// TIA Portal project "level-controle-factoryIO" (V17)

(* hardware
DEVICE "S71500/ET200MP-Station_1"  S7-1500 station
   slot 0: "Profilschiene_0"  6ES7 590-1***0-0AA0
   slot 1: "PLC_1"  CPU 1511-1 PN  6ES7 511-1AK00-0AB0  V1.8
   slot 2: "AI 8xU/I/RTD/TC ST_1"  AI 8xU/I/RTD/TC ST  6ES7 531-7KF00-0AB0  V2.0
   slot 3: "AI 8xU/I/RTD/TC ST_2"  AI 8xU/I/RTD/TC ST  6ES7 531-7KF00-0AB0  V2.0
   slot 4: "AI 8xU/I/RTD/TC ST_3"  AI 8xU/I/RTD/TC ST  6ES7 531-7KF00-0AB0  V2.0
   slot 5: "AI 8xU/I/RTD/TC ST_4"  AI 8xU/I/RTD/TC ST  6ES7 531-7KF00-0AB0  V2.0
   slot 6: "DI 16x24VDC BA_1"  DI 16x24VDC BA  6ES7 521-1BH10-0AA0  V1.0
DEVICE "HMI_1"  KTP900 Basic PN
   slot 0: "HMI_1"  KTP900 Basic PN  6AV2 123-2JB03-0AX0  17.0.0.0
   slot 1: "HMI_RT_1"  KTP900 Basic PN  6AV2 123-2JB03-0AX0  17.0.0.0
   slot 5: "HMI_1.IE_CP_1"  PROFINET Interface  17.0.0.0
      slot 1: "PROFINET Interface_1"  PROFINET Interface
         slot 1: "Port_1"  Port
*)

// ===== PLC "PLC_1"  CPU 1511-1 PN =====

VAR_GLOBAL   // PLC tag table "Standard-Variablentabelle"
   "Clock_Byte" AT %MB0 : Byte;
   "Clock_10Hz" AT %M0.0 : Bool;
   "Clock_5Hz" AT %M0.1 : Bool;
   "Clock_2.5Hz" AT %M0.2 : Bool;
   "Clock_2Hz" AT %M0.3 : Bool;
   "Clock_1.25Hz" AT %M0.4 : Bool;
   "Clock_1Hz" AT %M0.5 : Bool;
   "Clock_0.625Hz" AT %M0.6 : Bool;
   "Clock_0.5Hz" AT %M0.7 : Bool;
   "System_Byte" AT %MB1 : Byte;
   "FirstScan" AT %M1.0 : Bool;
   "DiagStatusUpdate" AT %M1.1 : Bool;
   "AlwaysTRUE" AT %M1.2 : Bool;
   "AlwaysFALSE" AT %M1.3 : Bool;
   "Tag_1" AT %M110.0 : Bool;
END_VAR

VAR_GLOBAL   // PLC tag table "Input"
   "I_LevelMeter" AT %ID30 : Real;
   "I_FlowMeter" AT %ID34 : Real;
   "I_FactoryRuning" AT %I0.0 : Bool;
END_VAR

VAR_GLOBAL   // PLC tag table "Output"
   "O_FillValve" AT %QD30 : Real;
   "O_DischargeValve" AT %QD34 : Real;
   "O_Empty" AT %Q0.0 : Bool;
END_VAR

// folder: 00_Visu

DATA_BLOCK "VisuData"   // DB9
{ S7_Optimized_Access := 'TRUE' }
VERSION : 0.1
   VAR
      Start : Bool;
      Stop : Bool;
      Empty : Bool;
      Controller : Int;
      RandomDisturbance : Int;
      SetPoint : Real;
      Outflow : Real;
      LevelMeterShow : Real;
      SetPointShow : Real;
      FillValveShow : Real;
      TopPump : Int;
      LowPump : Int;
      Status : Bool;
      default : Bool;
      finish_training : Int;
      factoryio_connect : Bool;
   END_VAR
BEGIN
END_DATA_BLOCK

// folder: 01_Convert

DATA_BLOCK "ConvertData"   // DB4
{ S7_Optimized_Access := 'TRUE' }
VERSION : 0.1
   VAR
      SetPoint10 : Real;
   END_VAR
BEGIN
END_DATA_BLOCK

// folder: 02_Controller

DATA_BLOCK "ControllerData"   // DB1
{ S7_Optimized_Access := 'TRUE' }
VERSION : 0.1
   VAR
      PID_Compact : Bool;
      Output_PID_Compact : Real;
      "IMC+PID" : Bool;
      rate : Real;
      hysteresis : Real;
      kp : Real;
      ki : Real;
      kd : Real;
   END_VAR
BEGIN
END_DATA_BLOCK

// folder: 02_Controller/NeuralNetwork

DATA_BLOCK "NeuroData"   // DB18
{ S7_Optimized_Access := 'TRUE' }
VERSION : 0.1
   VAR
      finish_measurment : Bool;
      disturbance : Real;
      PV : Real;
      MV : Real;
      SP : Real;
      stop_training_inw : Bool;
      stop_training_mod : Bool;
      epoka : Real;
      error_ep_m : Real;
      error_ep_i : Real;
      error_stop_m : Real;
      error_stop_i : Real;
      epoka_m : Real;
      epoka_i : Real;
      move : Bool;
      p_move : Bool;
      finish_training : Bool;
   END_VAR
BEGIN
END_DATA_BLOCK

// folder: System blocks/Program resources

DATA_BLOCK "PID_DB"   // DB2
{ S7_Optimized_Access := 'FALSE' }
VERSION : 0.1
// stored: InstanceOfName PID
"PID"
BEGIN
END_DATA_BLOCK

DATA_BLOCK "RandomDisturbance_DB"   // DB5
{ S7_Optimized_Access := 'TRUE' }
VERSION : 0.1
// stored: InstanceOfName RandomDisturbance
"RandomDisturbance"
BEGIN
END_DATA_BLOCK

DATA_BLOCK "RAMP_DB"   // DB6
{ S7_Optimized_Access := 'TRUE' }
VERSION : 0.1
// stored: InstanceOfName RAMP
"RAMP"
BEGIN
END_DATA_BLOCK

DATA_BLOCK "RegSugeno_DB"   // DB7
{ S7_Optimized_Access := 'TRUE' }
VERSION : 0.1
// stored: InstanceOfName Takagi-SugenoFuzzy-PI
"Takagi-SugenoFuzzy-PI"
BEGIN
END_DATA_BLOCK

DATA_BLOCK "Training_DB"   // DB10
{ S7_Optimized_Access := 'FALSE' }
VERSION : 0.1
// stored: InstanceOfName Training
"Training"
BEGIN
END_DATA_BLOCK

DATA_BLOCK "PID_DB_1"   // DB11
{ S7_Optimized_Access := 'FALSE' }
VERSION : 0.1
// stored: InstanceOfName PID
"PID"
BEGIN
END_DATA_BLOCK

DATA_BLOCK "Measurement_DB"   // DB12
{ S7_Optimized_Access := 'FALSE' }
VERSION : 0.1
// stored: InstanceOfName Measurement
"Measurement"
BEGIN
END_DATA_BLOCK

DATA_BLOCK "Object_DB"   // DB13
{ S7_Optimized_Access := 'FALSE' }
VERSION : 0.1
// stored: InstanceOfName Object
"Object"
BEGIN
END_DATA_BLOCK

DATA_BLOCK "Generator_DB"   // DB14
{ S7_Optimized_Access := 'FALSE' }
VERSION : 0.1
// stored: InstanceOfName Generator
"Generator"
BEGIN
END_DATA_BLOCK

DATA_BLOCK "IMC+PID_DB"   // DB15
{ S7_Optimized_Access := 'FALSE' }
VERSION : 0.1
// stored: InstanceOfName IMC+PID
"IMC+PID"
BEGIN
END_DATA_BLOCK

DATA_BLOCK "Model_DB"   // DB16
{ S7_Optimized_Access := 'FALSE' }
VERSION : 0.1
// stored: InstanceOfName Model
"Model"
BEGIN
END_DATA_BLOCK

DATA_BLOCK "Inversion_DB"   // DB17
{ S7_Optimized_Access := 'FALSE' }
VERSION : 0.1
// stored: InstanceOfName Inversion
"Inversion"
BEGIN
END_DATA_BLOCK

DATA_BLOCK "StartStop_DB"   // DB19
{ S7_Optimized_Access := 'TRUE' }
VERSION : 0.1
// stored: InstanceOfName StartStop
"StartStop"
BEGIN
END_DATA_BLOCK

DATA_BLOCK "On-Off_DB"   // DB20
{ S7_Optimized_Access := 'TRUE' }
VERSION : 0.1
// stored: InstanceOfName On-Off
"On-Off"
BEGIN
END_DATA_BLOCK

// folder: (top level)

FUNCTION "MHJ-PLC-Lab-Function-S71500" : Void   // FC9000, SCL
{ S7_Optimized_Access := 'TRUE' }
VERSION : 0.1
   VAR_TEMP
      Value : Byte;
      ForCounter : Int;
   END_VAR
   VAR CONSTANT
      Value_01_DW : DWord := 16#1223_5486;
      Value_02_DW : DWord := 16#A6C9_D1F5;
   END_VAR
BEGIN

   #Value:=PEEK(area := 16#82,
        dbNumber := 0,
        byteOffset := 511);
   #Value := #Value + 1;

   POKE(area := 16#82,
        dbNumber := 0,
        byteOffset := 511,
        value := #Value);

   POKE(area := 16#82,
        dbNumber := 0,
        byteOffset := 1016,
        value := #Value_01_DW);
   POKE(area := 16#82,
        dbNumber := 0,
        byteOffset := 1020,
        value := #Value_02_DW);

   FOR #ForCounter := 0 TO 63 DO
       #Value:=PEEK(area := 16#1,
            dbNumber := 0,
            byteOffset := #ForCounter);
       POKE(area := 16#81,
            dbNumber := 0,
            byteOffset := #ForCounter,
            value := #Value);
   END_FOR;
   #Value := PEEK(area := 16#1,
                  dbNumber := 0,
                  byteOffset := 512);
   POKE(area := 16#82,
        dbNumber := 0,
        byteOffset := 512,
        value := #Value);
END_FUNCTION

ORGANIZATION_BLOCK "Main"   // OB1, LAD, ProgramCycle
TITLE = "Main Program Sweep (Cycle)"
{ S7_Optimized_Access := 'TRUE' }
VERSION : 0.1
   VAR_INPUT
      Initial_Call : Bool;   // Initial call of this OB
      Remanence : Bool;   // =True, if remanent data are available
   END_VAR
BEGIN

REGION Network 1: Call: MHJ-PLC-Lab-Function-S71500
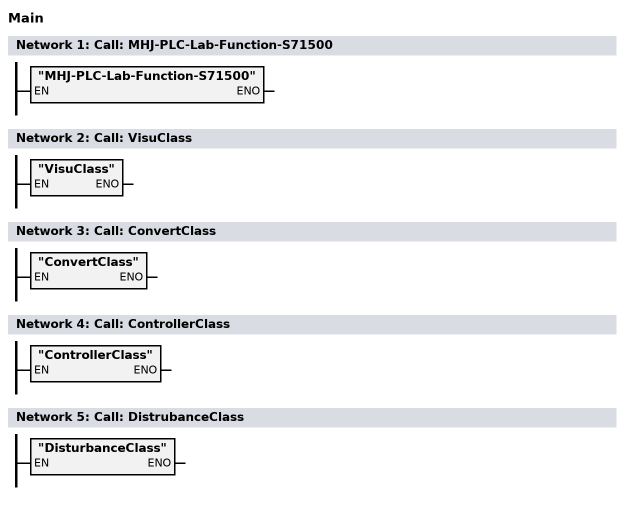
   RUNG wire#powerrail
      "MHJ-PLC-Lab-Function-S71500"()
   END_RUNG
   // the same network as SCL:
   "MHJ-PLC-Lab-Function-S71500"();
END_REGION

REGION Network 2: Call: VisuClass
   RUNG wire#powerrail
      "VisuClass"()
   END_RUNG
   // the same network as SCL:
   "VisuClass"();
END_REGION

REGION Network 3: Call: ConvertClass
   RUNG wire#powerrail
      "ConvertClass"()
   END_RUNG
   // the same network as SCL:
   "ConvertClass"();
END_REGION

REGION Network 4: Call: ControllerClass
   RUNG wire#powerrail
      "ControllerClass"()
   END_RUNG
   // the same network as SCL:
   "ControllerClass"();
END_REGION

REGION Network 5: Call: DistrubanceClass
   RUNG wire#powerrail
      "DisturbanceClass"()
   END_RUNG
   // the same network as SCL:
   "DisturbanceClass"();
END_REGION
END_ORGANIZATION_BLOCK

ORGANIZATION_BLOCK "Startup"   // OB100, LAD, Startup
TITLE = "Complete Restart"
{ S7_Optimized_Access := 'TRUE' }
VERSION : 0.1
   VAR_INPUT
      LostRetentive : Bool;   // True if retentive data are lost
      LostRTC : Bool;   // True if date and time are lost
   END_VAR
BEGIN

REGION Network 1: Call: StartupValues
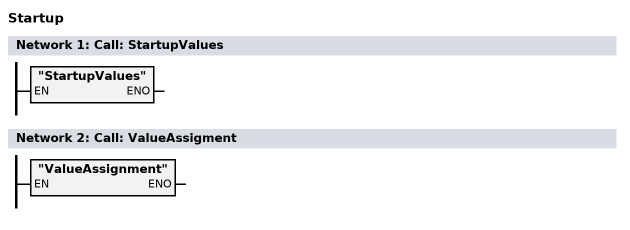
   RUNG wire#powerrail
      "StartupValues"()
   END_RUNG
   // the same network as SCL:
   "StartupValues"();
END_REGION

REGION Network 2: Call: ValueAssigment
   RUNG wire#powerrail
      "ValueAssignment"()
   END_RUNG
   // the same network as SCL:
   "ValueAssignment"();
END_REGION
END_ORGANIZATION_BLOCK

// folder: 00_Visu

FUNCTION "ShowPompOn" : Void   // FC6, LAD
TITLE = ShowPompOn
{ S7_Optimized_Access := 'TRUE' }
VERSION : 0.1
   VAR_TEMP   // added for the SCL form of the ladder/FBD networks
      _w1 : Bool;
   END_VAR
BEGIN

REGION Network 1: Move: TopPump
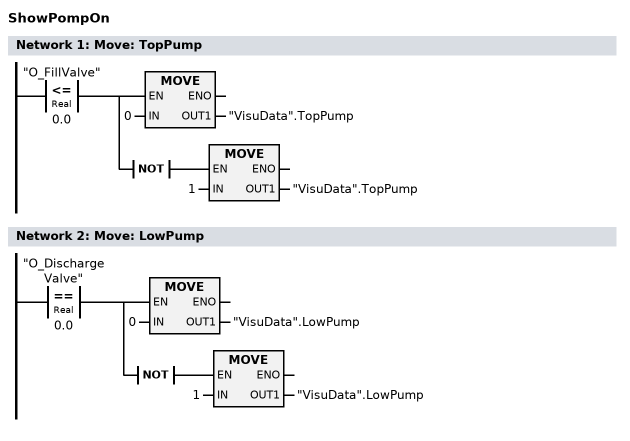
   RUNG wire#powerrail
      { S7_Templates := "SrcType := Real" } LE_Contact(in1 := "O_FillValve", in2 := 0.0)
      wire#w1
      Move(in := 0, out1 => "VisuData".TopPump)
   END_RUNG
   RUNG wire#w1
      Not()
      Move(in := 1, out1 => "VisuData".TopPump)
   END_RUNG
   // the same network as SCL:
   #_w1 := "O_FillValve" <= 0.0;
   IF #_w1 THEN "VisuData".TopPump := 0; END_IF;
   IF NOT #_w1 THEN "VisuData".TopPump := 1; END_IF;
END_REGION

REGION Network 2: Move: LowPump
   RUNG wire#powerrail
      { S7_Templates := "SrcType := Real" } EQ_Contact(in1 := "O_DischargeValve", in2 := 0.0)
      wire#w1
      Move(in := 0, out1 => "VisuData".LowPump)
   END_RUNG
   RUNG wire#w1
      Not()
      Move(in := 1, out1 => "VisuData".LowPump)
   END_RUNG
   // the same network as SCL:
   #_w1 := "O_DischargeValve" = 0.0;
   IF #_w1 THEN "VisuData".LowPump := 0; END_IF;
   IF NOT #_w1 THEN "VisuData".LowPump := 1; END_IF;
END_REGION
END_FUNCTION

FUNCTION "VisuClass" : Void   // FC8, LAD
TITLE = VisuClass
{ S7_Optimized_Access := 'TRUE' }
VERSION : 0.1
BEGIN

REGION Network 1: Call: StartStop
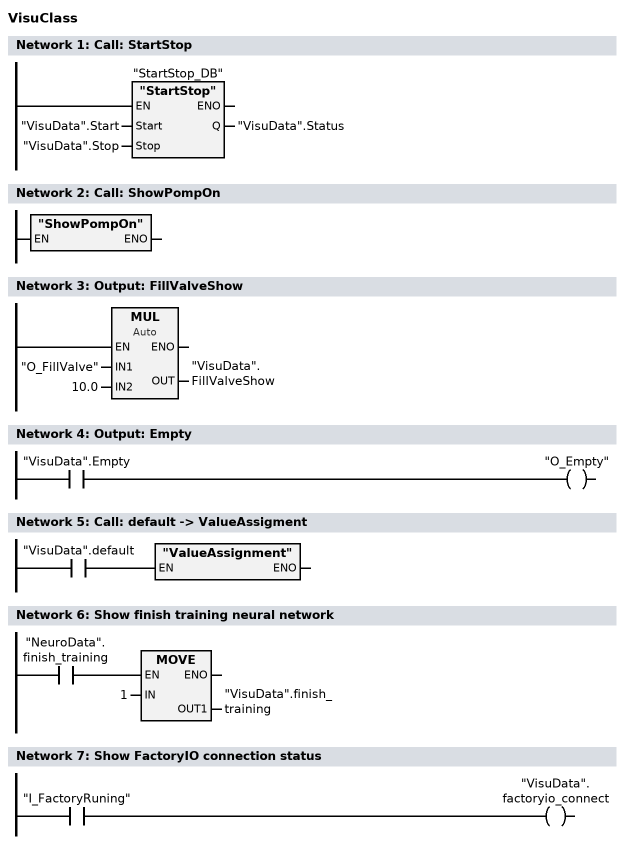
   RUNG wire#powerrail
      "StartStop_DB"(Start := "VisuData".Start, Stop := "VisuData".Stop, Q => "VisuData".Status)
   END_RUNG
   // the same network as SCL:
   "StartStop_DB"(Start := "VisuData".Start, Stop := "VisuData".Stop, Q => "VisuData".Status);   // "StartStop"
END_REGION

REGION Network 2: Call: ShowPompOn
   RUNG wire#powerrail
      "ShowPompOn"()
   END_RUNG
   // the same network as SCL:
   "ShowPompOn"();
END_REGION

REGION Network 3: Output: FillValveShow
   RUNG wire#powerrail
      Mul(in1 := "O_FillValve", in2 := 10.0, out => "VisuData".FillValveShow)
   END_RUNG
   // the same network as SCL:
   "VisuData".FillValveShow := "O_FillValve" * 10.0;
END_REGION

REGION Network 4: Output: Empty
   RUNG wire#powerrail
      Contact( "VisuData".Empty )
      Coil( "O_Empty" )
   END_RUNG
   // the same network as SCL:
   "O_Empty" := "VisuData".Empty;
END_REGION

REGION Network 5: Call: default -> ValueAssigment
   RUNG wire#powerrail
      Contact( "VisuData".default )
      "ValueAssignment"()
   END_RUNG
   // the same network as SCL:
   IF "VisuData".default THEN "ValueAssignment"(); END_IF;
END_REGION

REGION Network 6: Show finish training neural network
   RUNG wire#powerrail
      Contact( "NeuroData".finish_training )
      Move(in := 1, out1 => "VisuData".finish_training)
   END_RUNG
   // the same network as SCL:
   IF "NeuroData".finish_training THEN "VisuData".finish_training := 1; END_IF;
END_REGION

REGION Network 7: Show FactoryIO connection status
   RUNG wire#powerrail
      Contact( "I_FactoryRuning" )
      Coil( "VisuData".factoryio_connect )
   END_RUNG
   // the same network as SCL:
   "VisuData".factoryio_connect := "I_FactoryRuning";
END_REGION
END_FUNCTION

// folder: 01_Convert

FUNCTION "ConvertClass" : Void   // FC3, LAD
TITLE = ConvertClass
{ S7_Optimized_Access := 'TRUE' }
VERSION : 0.1
   VAR_TEMP
      Output_PID_Real : Real;
      PV : Real;
      SP : Real;
      SPRamp : Real;
   END_VAR
BEGIN

REGION Network 1: Convert SetPoint: 0-300 -> 0-10
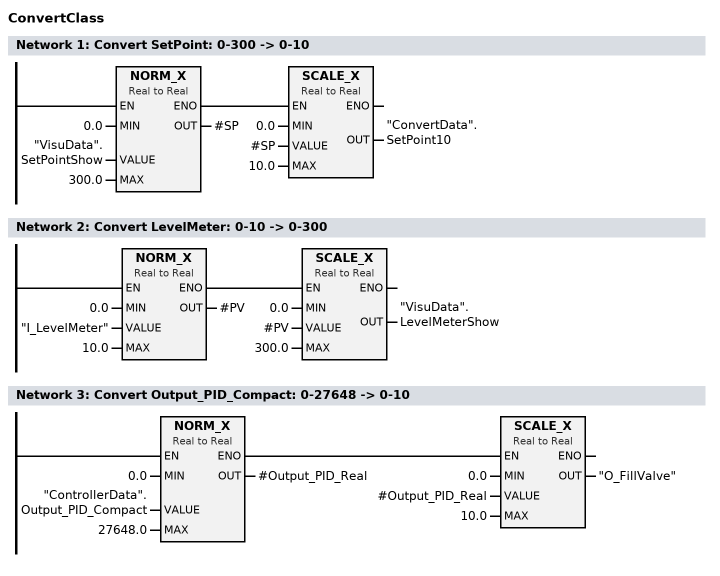
   RUNG wire#powerrail
      { S7_Templates := "[SrcType := Real, DestType := Real]" } Normalize(min := 0.0, value := "VisuData".SetPointShow, max := 300.0, out => #SP)
      { S7_Templates := "[SrcType := Real, DestType := Real]" } Scale(min := 0.0, value := #SP, max := 10.0, out => "ConvertData".SetPoint10)
   END_RUNG
   // the same network as SCL:
   #SP := NORM_X(MIN := 0.0, VALUE := "VisuData".SetPointShow, MAX := 300.0);
   "ConvertData".SetPoint10 := SCALE_X(MIN := 0.0, VALUE := #SP, MAX := 10.0);
END_REGION

REGION Network 2: Convert LevelMeter: 0-10 -> 0-300
   RUNG wire#powerrail
      { S7_Templates := "[SrcType := Real, DestType := Real]" } Normalize(min := 0.0, value := "I_LevelMeter", max := 10.0, out => #PV)
      { S7_Templates := "[SrcType := Real, DestType := Real]" } Scale(min := 0.0, value := #PV, max := 300.0, out => "VisuData".LevelMeterShow)
   END_RUNG
   // the same network as SCL:
   #PV := NORM_X(MIN := 0.0, VALUE := "I_LevelMeter", MAX := 10.0);
   "VisuData".LevelMeterShow := SCALE_X(MIN := 0.0, VALUE := #PV, MAX := 300.0);
END_REGION

REGION Network 3: Convert Output_PID_Compact: 0-27648 -> 0-10
   RUNG wire#powerrail
      { S7_Templates := "[SrcType := Real, DestType := Real]" } Normalize(min := 0.0, value := "ControllerData".Output_PID_Compact, max := 27648.0, out => #Output_PID_Real)
      { S7_Templates := "[SrcType := Real, DestType := Real]" } Scale(min := 0.0, value := #Output_PID_Real, max := 10.0, out => "O_FillValve")
   END_RUNG
   // the same network as SCL:
   #Output_PID_Real := NORM_X(MIN := 0.0, VALUE := "ControllerData".Output_PID_Compact, MAX := 27648.0);
   "O_FillValve" := SCALE_X(MIN := 0.0, VALUE := #Output_PID_Real, MAX := 10.0);
END_REGION
END_FUNCTION

// folder: 02_Controller

FUNCTION_BLOCK "Takagi-SugenoFuzzy-PI"   // FB7, SCL
{ S7_Optimized_Access := 'TRUE' }
VERSION : 0.1
   VAR_INPUT
      PV : Real;
      SP : Real;
   END_VAR
   VAR_OUTPUT
      MV : Real;
   END_VAR
   VAR
      n_e : Real;
      i_e : Real;
      ni_e : Real;
   END_VAR
   VAR_TEMP
      "e" : Real;
      u : Real;
      sp_M_e : Real;
      sp_S_e : Real;
      sp_D_e : Real;
      sp_M_ie : Real;
      sp_S_ie : Real;
      sp_D_ie : Real;
      pz1 : Real;
      pz2 : Real;
      pz3 : Real;
      pz4 : Real;
      pz5 : Real;
      pz6 : Real;
      pz7 : Real;
      pz8 : Real;
      pz9 : Real;
   END_VAR
BEGIN
   #n_e:=5.0;
   #ni_e:=0.25;

   #e:=#SP-#PV;
   #e:=#n_e*#e;
   IF #e>10.0 THEN
       #e := 10.0;
   ELSIF #e<-10.0 THEN
     #e:=-10.0;
   END_IF;

   #i_e:=#i_e+#e;
   #i_e:=#ni_e*#i_e;
   IF #i_e>10.0 THEN
     #i_e:=10.0;
   ELSIF #i_e<-10.0 THEN
     #i_e:=-10.0;
   END_IF;

   IF #e<0.0 THEN
     #sp_M_e:=(#e)/-10.0;
     #sp_S_e:=(#e)/10.0+1.0;
     #sp_D_e:=0.0;
   ELSIF #e>0.0 THEN
     #sp_D_e:=(#e)/10.0;
     #sp_S_e:=(#e)/-10.0+1.0;
     #sp_M_e:=0.0;
   ELSE
     #sp_M_e:=0.0;
     #sp_D_e:=0.0;
     #sp_S_e:=1.0;
   END_IF;

   IF #i_e<0.0 THEN
     #sp_M_ie:=(#i_e)/-10.0;
     #sp_S_ie:=(#i_e)/10.0+1.0; //jw.
     #sp_D_ie:=0.0;
   ELSIF #i_e>0.0 THEN
     #sp_D_ie:=(#i_e)/10.0;
     #sp_S_ie:=(#i_e)/-10.0+1.0;//jw.
     #sp_M_ie:=0.0;
   ELSE
     #sp_M_ie:=0.0;
     #sp_D_ie:=0.0;
     #sp_S_ie:=1.0;
   END_IF;

   #pz1:=MIN(IN1:=#sp_M_e, IN2:=#sp_M_ie); 
   #pz2:=MIN(IN1:=#sp_S_e, IN2:=#sp_M_ie);
   #pz3:=MIN(IN1:=#sp_D_e, IN2:=#sp_M_ie);
   #pz4:=MIN(IN1:=#sp_M_e, IN2:=#sp_S_ie);
   #pz5:=MIN(IN1:=#sp_S_e, IN2:=#sp_S_ie);
   #pz6:=MIN(IN1:=#sp_D_e, IN2:=#sp_S_ie);
   #pz7:=MIN(IN1:=#sp_M_e, IN2:=#sp_D_ie);
   #pz8:=MIN(IN1:=#sp_S_e, IN2:=#sp_D_ie);
   #pz9:=MIN(IN1:=#sp_D_e, IN2:=#sp_D_ie);

    #u:=(#pz1*0.0+#pz2*0.0+#pz3*5.0+#pz4*0.0+#pz5*5.0
                       +#pz6*10.0+#pz7*5.0++#pz8*10.0++#pz9*10.0)
                       /(#pz1+#pz2+#pz3+#pz4+#pz5+#pz6+#pz7+#pz8+#pz9);

   IF #u>10.0 THEN
     #u:=10.0;
   END_IF;

   IF #u < 5.0 AND #u > -5.0 THEN
       #u := 0;
   END_IF;

   IF #u < -10.0 THEN
       #u := -10.0;
   END_IF;

   #MV := #u;
END_FUNCTION_BLOCK

FUNCTION_BLOCK "RAMP"   // FB8, LAD
TITLE = RAMP
{ S7_Optimized_Access := 'TRUE' }
VERSION : 0.1
   VAR_INPUT
      SetPoint : Real;
      Rate : Real;
      Reset : Bool;
   END_VAR
   VAR_OUTPUT
      OUT : Real := 0.0;
   END_VAR
   VAR
      TON_1 : TON_TIME;
      RateDIV : Real;
      Q : Bool;
   END_VAR
   VAR_TEMP   // added for the SCL form of the ladder/FBD networks
      _w1 : Bool;
   END_VAR
BEGIN

REGION Network 1: DIV: Rate/10
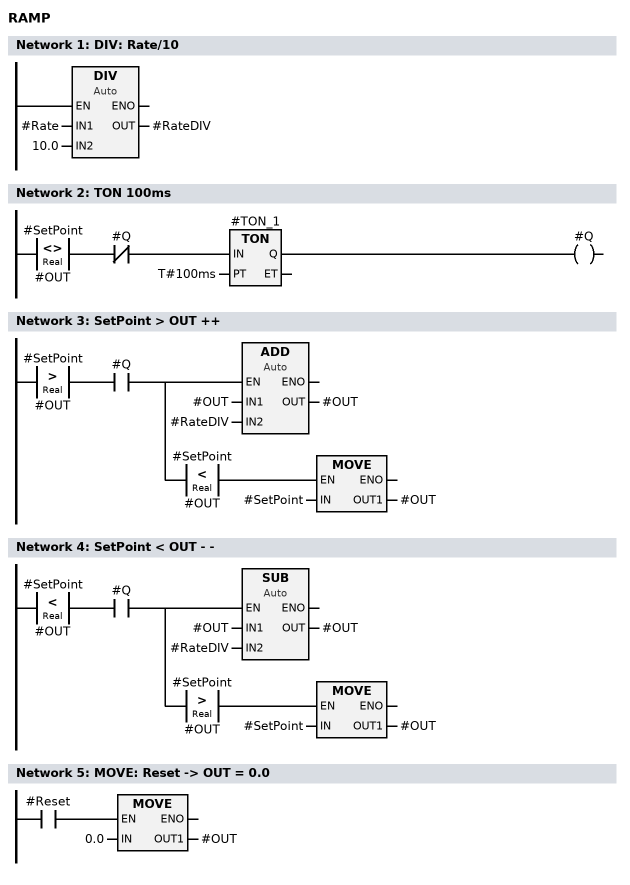
   RUNG wire#powerrail
      Div(in1 := #Rate, in2 := 10.0, out => #RateDIV)
   END_RUNG
   // the same network as SCL:
   #RateDIV := #Rate / 10.0;
END_REGION

REGION Network 2: TON 100ms
   #TON_1(IN := (#SetPoint <> #OUT) AND NOT #Q, PT := T#100ms);   // TON
   #Q := #TON_1.Q;
END_REGION

REGION Network 3: SetPoint > OUT ++
   RUNG wire#powerrail
      { S7_Templates := "SrcType := Real" } GT_Contact(in1 := #SetPoint, in2 := #OUT)
      Contact( #Q )
      wire#w1
      Add(in1 := #OUT, in2 := #RateDIV, out => #OUT)
   END_RUNG
   RUNG wire#w1
      { S7_Templates := "SrcType := Real" } LT_Contact(in1 := #SetPoint, in2 := #OUT)
      Move(in := #SetPoint, out1 => #OUT)
   END_RUNG
   // the same network as SCL:
   #_w1 := (#SetPoint > #OUT) AND #Q;
   IF #_w1 THEN #OUT := #OUT + #RateDIV; END_IF;
   IF #_w1 AND (#SetPoint < #OUT) THEN #OUT := #SetPoint; END_IF;
END_REGION

REGION Network 4: SetPoint < OUT - -
   RUNG wire#powerrail
      { S7_Templates := "SrcType := Real" } LT_Contact(in1 := #SetPoint, in2 := #OUT)
      Contact( #Q )
      wire#w1
      Sub(in1 := #OUT, in2 := #RateDIV, out => #OUT)
   END_RUNG
   RUNG wire#w1
      { S7_Templates := "SrcType := Real" } GT_Contact(in1 := #SetPoint, in2 := #OUT)
      Move(in := #SetPoint, out1 => #OUT)
   END_RUNG
   // the same network as SCL:
   #_w1 := (#SetPoint < #OUT) AND #Q;
   IF #_w1 THEN #OUT := #OUT - #RateDIV; END_IF;
   IF #_w1 AND (#SetPoint > #OUT) THEN #OUT := #SetPoint; END_IF;
END_REGION

REGION Network 5: MOVE: Reset -> OUT = 0.0
   RUNG wire#powerrail
      Contact( #Reset )
      Move(in := 0.0, out1 => #OUT)
   END_RUNG
   // the same network as SCL:
   IF #Reset THEN #OUT := 0.0; END_IF;
END_REGION
END_FUNCTION_BLOCK

FUNCTION_BLOCK "PID"   // FB9, SCL
{ S7_Optimized_Access := 'FALSE' }
VERSION : 0.1
   VAR_INPUT
      SP : Real;
      PV : Real;
      MV : Real;
      kp : Real;
      ki : Real;
      kd : Real;
   END_VAR
   VAR_OUTPUT
      MV_PID : Real;
   END_VAR
   VAR
      ep : Array[0..1] of Real;
      de : Real;
      suma_ep : Real;
   END_VAR
BEGIN
   #ep[0]:=#SP-#PV;

   IF (ABS(#ep[0]))<(ABS(#SP)) THEN
     #de:=#ep[0]-#ep[1];                                   

     IF #MV<10.0 THEN
       IF #MV>-10.0 THEN      
         #suma_ep:=#suma_ep+#ep[0];
       END_IF;
     END_IF;

     #MV_PID:=#kp*#ep[0] + #ki*#suma_ep + #kd*#de;  

     IF #MV_PID > 10.0 THEN
         #MV_PID := 10.0;
     END_IF;

     IF #MV_PID < -10.0 THEN
         #MV_PID := -10.0;
     END_IF;

     #ep[1]:=#ep[0];

   ELSE                      
     #ep[1]:=0.0;
     #suma_ep:=0.0;

   END_IF;
END_FUNCTION_BLOCK

FUNCTION_BLOCK "StartStop"   // FB11, LAD
TITLE = StartStop
{ S7_Optimized_Access := 'TRUE' }
VERSION : 0.1
   VAR_INPUT
      Start : Bool;
      Stop : Bool;
   END_VAR
   VAR_OUTPUT
      Q : Bool;
   END_VAR
   VAR
      statSR : Bool;
      statRisEdge : Bool;
   END_VAR
   VAR_TEMP   // added for the SCL form of the ladder/FBD networks
      _w1 : Bool;
   END_VAR
BEGIN

REGION Network 1: P_Trig && SR
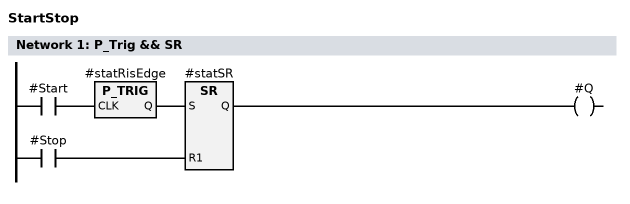
   RUNG wire#powerrail
      Contact( #Start )
      P_Trig( #statRisEdge )
      S_SR(operand := #statSR, r1 := wire#w1)
      Coil( #Q )
   END_RUNG
   RUNG wire#powerrail
      Contact( #Stop )
   END_RUNG wire#w1
   // the same network as SCL:
   #_w1 := #Start AND NOT #statRisEdge;   // rising edge
   #statRisEdge := #Start;
   IF #_w1 THEN
       #statSR := TRUE;   // SR flip-flop
   END_IF;
   IF #Stop THEN #statSR := FALSE; END_IF;
   #Q := #statSR;
END_REGION
END_FUNCTION_BLOCK

FUNCTION_BLOCK "On-Off"   // FB12, SCL
{ S7_Optimized_Access := 'TRUE' }
VERSION : 0.1
   VAR_INPUT
      SetPoint : Real;   // Real
      Hysteresis : Real;   // Real
      PV : Real;   // Real
   END_VAR
   VAR_OUTPUT
      MV : Real;   // Real
   END_VAR
   VAR
      UpperLimit : Real;
      LowerLimit : Real;
   END_VAR
BEGIN
   #UpperLimit := #SetPoint + #Hysteresis / 2;
   #LowerLimit := #SetPoint - #Hysteresis / 2;

   IF #PV > #UpperLimit THEN
       #MV := -10.0;
       IF #PV = #LowerLimit THEN
           #MV := 0.0;
       END_IF;
   END_IF;


   IF #PV < #LowerLimit THEN
       #MV := 10.0;

       IF #PV = #UpperLimit THEN
           #MV := 0.0;
       END_IF;
   END_IF;
END_FUNCTION_BLOCK

FUNCTION "ControllerClass" : Void   // FC2, LAD
TITLE = ControllerClass
{ S7_Optimized_Access := 'TRUE' }
VERSION : 0.1
   VAR_TEMP
      MV : Real;
      SP : Real;
   END_VAR
   VAR_TEMP   // added for the SCL form of the ladder/FBD networks
      _w1 : Bool;
   END_VAR
BEGIN

REGION Network 1: Call: Ramp
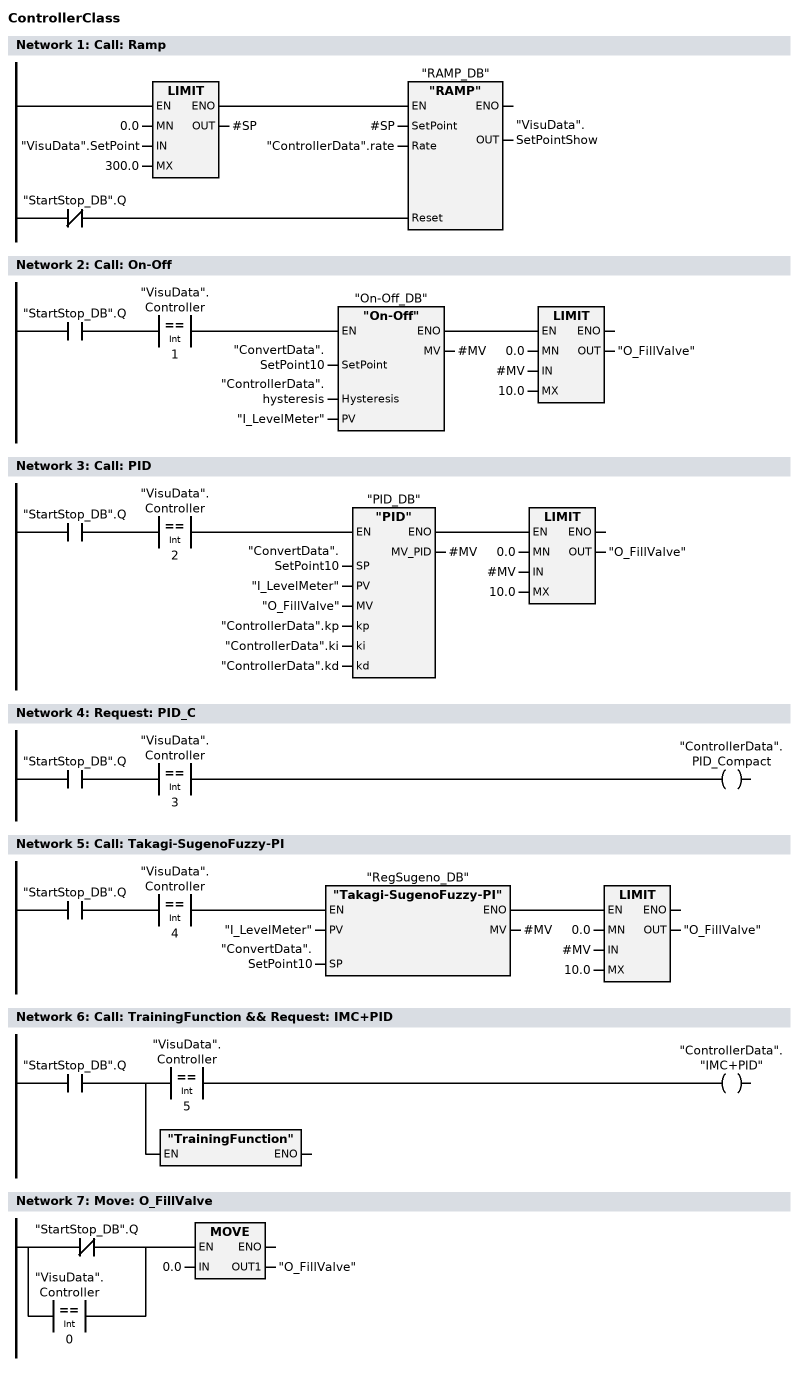
   #SP := LIMIT(MN := 0.0, IN := "VisuData".SetPoint, MX := 300.0);
   "RAMP_DB"(SetPoint := #SP,   // "RAMP"
             Rate := "ControllerData".rate,
             Reset := NOT "StartStop_DB".Q,
             OUT => "VisuData".SetPointShow);
END_REGION

REGION Network 2: Call: On-Off
   "On-Off_DB"(EN := "StartStop_DB".Q AND ("VisuData".Controller = 1),   // "On-Off"
               SetPoint := "ConvertData".SetPoint10,
               Hysteresis := "ControllerData".hysteresis,
               PV := "I_LevelMeter",
               MV => #MV,
               ENO => #_w1);
   IF #_w1 THEN "O_FillValve" := LIMIT(MN := 0.0, IN := #MV, MX := 10.0); END_IF;
END_REGION

REGION Network 3: Call: PID
   "PID_DB"(EN := "StartStop_DB".Q AND ("VisuData".Controller = 2),   // "PID"
            SP := "ConvertData".SetPoint10,
            PV := "I_LevelMeter",
            MV := "O_FillValve",
            kp := "ControllerData".kp,
            ki := "ControllerData".ki,
            kd := "ControllerData".kd,
            MV_PID => #MV,
            ENO => #_w1);
   IF #_w1 THEN "O_FillValve" := LIMIT(MN := 0.0, IN := #MV, MX := 10.0); END_IF;
END_REGION

REGION Network 4: Request: PID_C
   RUNG wire#powerrail
      Contact( "StartStop_DB".Q )
      { S7_Templates := "SrcType := Int" } EQ_Contact(in1 := "VisuData".Controller, in2 := 3)
      Coil( "ControllerData".PID_Compact )
   END_RUNG
   // the same network as SCL:
   "ControllerData".PID_Compact := "StartStop_DB".Q AND ("VisuData".Controller = 3);
END_REGION

REGION Network 5: Call: Takagi-SugenoFuzzy-PI
   "RegSugeno_DB"(EN := "StartStop_DB".Q AND ("VisuData".Controller = 4),   // "Takagi-SugenoFuzzy-PI"
                  PV := "I_LevelMeter",
                  SP := "ConvertData".SetPoint10,
                  MV => #MV,
                  ENO => #_w1);
   IF #_w1 THEN "O_FillValve" := LIMIT(MN := 0.0, IN := #MV, MX := 10.0); END_IF;
END_REGION

REGION Network 6: Call: TrainingFunction && Request: IMC+PID
   RUNG wire#powerrail
      Contact( "StartStop_DB".Q )
      wire#w1
      { S7_Templates := "SrcType := Int" } EQ_Contact(in1 := "VisuData".Controller, in2 := 5)
      Coil( "ControllerData"."IMC+PID" )
   END_RUNG
   RUNG wire#w1
      "TrainingFunction"()
   END_RUNG
   // the same network as SCL:
   "ControllerData"."IMC+PID" := "StartStop_DB".Q AND ("VisuData".Controller = 5);
   IF "StartStop_DB".Q THEN "TrainingFunction"(); END_IF;
END_REGION

REGION Network 7: Move: O_FillValve
   RUNG wire#powerrail
      I_Contact( "StartStop_DB".Q )
      wire#w1
      Move(in := 0.0, out1 => "O_FillValve")
   END_RUNG
   RUNG wire#powerrail
      { S7_Templates := "SrcType := Int" } EQ_Contact(in1 := "VisuData".Controller, in2 := 0)
   END_RUNG wire#w1
   // the same network as SCL:
   IF NOT "StartStop_DB".Q OR ("VisuData".Controller = 0) THEN "O_FillValve" := 0.0; END_IF;
END_REGION
END_FUNCTION

FUNCTION "ValueAssignment" : Void   // FC9, LAD
TITLE = ValueAssignment
{ S7_Optimized_Access := 'TRUE' }
VERSION : 0.1
BEGIN

REGION Network 1: Move: rate
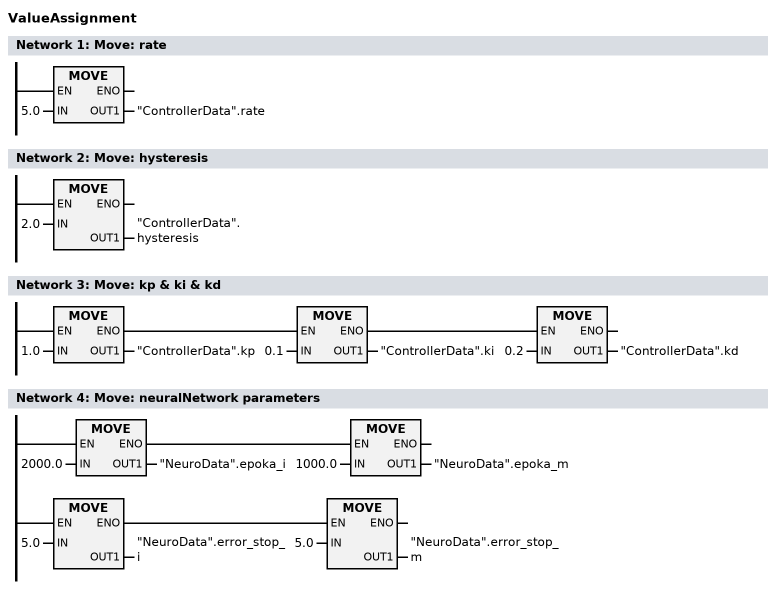
   RUNG wire#powerrail
      Move(in := 5.0, out1 => "ControllerData".rate)
   END_RUNG
   // the same network as SCL:
   "ControllerData".rate := 5.0;
END_REGION

REGION Network 2: Move: hysteresis
   RUNG wire#powerrail
      Move(in := 2.0, out1 => "ControllerData".hysteresis)
   END_RUNG
   // the same network as SCL:
   "ControllerData".hysteresis := 2.0;
END_REGION

REGION Network 3: Move: kp & ki & kd
   RUNG wire#powerrail
      Move(in := 1.0, out1 => "ControllerData".kp)
      Move(in := 0.1, out1 => "ControllerData".ki)
      Move(in := 0.2, out1 => "ControllerData".kd)
   END_RUNG
   // the same network as SCL:
   "ControllerData".kp := 1.0;
   "ControllerData".ki := 0.1;
   "ControllerData".kd := 0.2;
END_REGION

REGION Network 4: Move: neuralNetwork parameters
   RUNG wire#powerrail
      Move(in := 2000.0, out1 => "NeuroData".epoka_i)
      Move(in := 1000.0, out1 => "NeuroData".epoka_m)
   END_RUNG
   RUNG wire#powerrail
      Move(in := 5.0, out1 => "NeuroData".error_stop_i)
      Move(in := 5.0, out1 => "NeuroData".error_stop_m)
   END_RUNG
   // the same network as SCL:
   "NeuroData".epoka_i := 2000.0;
   "NeuroData".epoka_m := 1000.0;
   "NeuroData".error_stop_i := 5.0;
   "NeuroData".error_stop_m := 5.0;
END_REGION
END_FUNCTION

ORGANIZATION_BLOCK "PID_C"   // OB30, LAD, CyclicInterrupt
{ S7_Optimized_Access := 'TRUE' }
VERSION : 0.1
   VAR_INPUT
      Initial_Call : Bool;   // Initial call of this OB
      Event_Count : Int;   // Events discarded
   END_VAR
BEGIN

REGION Network 1: PID_Compact
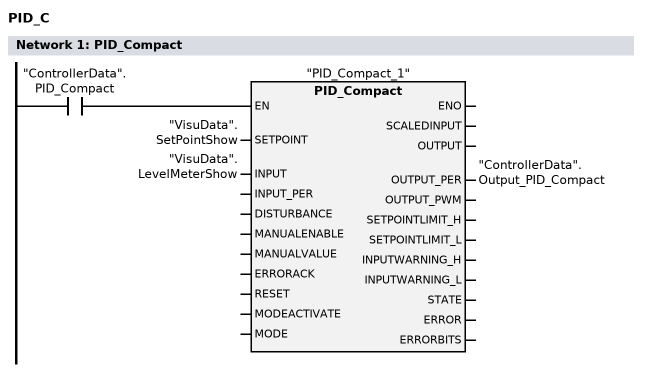
   IF "ControllerData".PID_Compact THEN
       "PID_Compact_1"(Setpoint := "VisuData".SetPointShow,   // PID_Compact
                       Input := "VisuData".LevelMeterShow,
                       Output_PER => "ControllerData".Output_PID_Compact);
   END_IF;
END_REGION
END_ORGANIZATION_BLOCK

// folder: 02_Controller/NeuralNetwork

FUNCTION_BLOCK "Measurement"   // FB1, SCL
{ S7_Optimized_Access := 'FALSE' }
VERSION : 0.1
   VAR_INPUT
      y : Real;   // zmierzona wartość odpowiedzi
   END_VAR
   VAR_OUTPUT
      r : Real;   // sygnał wysyłany na obiekt
      finish : Bool;   // sygnalizacja zakończenia pomiaru
   END_VAR
   VAR
      r_array : Array[0..249] of Real;   // zapisywany wektor wzorcowy wejść
      y_array : Array[0..249] of Real;   // zapisywany wektor wzorcowy odpowiedzi
      i : Int;   // iteracja, zmienna pomocnicza
   END_VAR
BEGIN
   IF #i=0 THEN
       #r:=#r_array[#i];
   END_IF;

   IF #i>0 THEN
       IF #i<250 THEN
           #y_array[#i-1]:=#y;
           #r:=#r_array[#i];
       END_IF;
   END_IF;

   IF #i=250 THEN
       #y_array[#i-1]:=#y;
       #finish:=true;
       #r:=0.0;
   END_IF;

   #i:=#i+1;
END_FUNCTION_BLOCK

FUNCTION_BLOCK "Training"   // FB2, SCL
{ S7_Optimized_Access := 'FALSE' }
VERSION : 0.1
   VAR_INPUT
      error_stop_m : Real;   // wartość błędu zatrzymująca uczenie modelu
      error_stop_i : Real;   // wartość błędu zatrzymująca uczenie inwersji
      epoch_stop_m : Real;   // numer epoki zatrzymujący uczenie modelu
      epoch_stop_i : Real;   // numer epoki zatrzymujący uczenie inwersji
      training_m : Bool;   // jeżeli 1 - ucz model
      training_i : Bool;   // jeżeli 1 - ucz inwersje
   END_VAR
   VAR_OUTPUT
      error_ep_m : Real;   // błąd epoki uczenia modelu
      error_ep_i : Real;   // błąd epoki uczenia inwersji
      stop_m : Bool;   // ukończono uczenie modelu
      stop_i : Bool;   // ukończono uczenie inwersji
   END_VAR
   VAR_IN_OUT
      epoch : Real;   // numer epoki
   END_VAR
   VAR
      i : Int;   // zmienna pomocnicza
      long : Int;   // zmienna pomocnicza
      s : Array[0..7] of Real;   // tablica sum ważonych neuronów warstwy ukrytej
      o : Array[0..7] of Real;   // tablica wyjść neuronów warstwy ukrytej
      s2 : Real;   // suma ważona warstwy wyjściowej
      e2 : Real;   // błąd na wyjściu sieci
      "e" : Array[0..7] of Real;   // błędy propagowane
      x_m : Array[0..5] of Real;   // wejścia sieci modelu
      x_i : Array[0..5] of Real;   // wejścia sieci inwersji
      n_m : Real;   // współczynnik prędkości uczenia sieci modelu
      n_i : Real;   // współczynnik prędkości uczenia sieci inwersji
   END_VAR
BEGIN
   #n_m:=0.005;
   #n_i:=0.001;

   IF #training_m=true THEN
     FOR #long:=0 TO 249 DO
       IF #long=0 THEN
         #x_m[2]:=0.0;         // x(k-2)
         #x_m[1]:=0.0;         // x(k-1)
         #x_m[0]:="Measurement_DB".r_array[#long];  // x(k)
         #x_m[5]:=0.0;         // y(k-3)
         #x_m[4]:=0.0;         // y(k-2)
         #x_m[3]:=0.0;         // y(k-1)
       ELSE
         #x_m[2]:=#x_m[1];     // x(k-2)             
         #x_m[1]:=#x_m[0];     // x(k-1)
         #x_m[0]:="Measurement_DB".r_array[#long];  // x(k)
         #x_m[5]:=#x_m[4];     // y(k-3)
         #x_m[4]:=#x_m[3];     // y(k-2)
         #x_m[3]:="Measurement_DB".y_array[#long-1]; // y(k-1)
       END_IF;

       FOR #i:=0 TO "Model_DB".N-1 DO 
          #s[#i]:=#x_m[0]*"Model_DB".w1_1[#i] + #x_m[1]*"Model_DB".w1_2[#i] + #x_m[2]*"Model_DB".w1_3[#i] + #x_m[3]*"Model_DB".w1_4[#i]; 
          #s[#i]:=#s[#i] + #x_m[4]*"Model_DB".w1_5[#i] + #x_m[5]*"Model_DB".w1_6[#i] + "Model_DB".bias[#i];
          #o[#i]:=(1.0-EXP(-#s[#i]))/(1.0+EXP(-#s[#i]));
       END_FOR;

       #s2:=0.0;
       FOR #i:=0 TO "Model_DB".N-1 DO
           #s2:=#s2+#o[#i]*"Model_DB".w_2[#i];
       END_FOR;
       #s2:=#s2+"Model_DB".bias2;

       #e2:="Measurement_DB".y_array[#long]-#s2;                                   

       FOR #i:=0 TO "Model_DB".N-1 DO
           #e[#i]:=#e2*"Model_DB".w_2[#i]*(1.0-(#o[#i]*#o[#i]));
       END_FOR;

       FOR #i:=0 TO "Model_DB".N-1 DO                                     
           "Model_DB".w1_1[#i]:="Model_DB".w1_1[#i]+#n_m*#e[#i]*#x_m[0];
           "Model_DB".w1_2[#i]:="Model_DB".w1_2[#i]+#n_m*#e[#i]*#x_m[1];
           "Model_DB".w1_3[#i]:="Model_DB".w1_3[#i]+#n_m*#e[#i]*#x_m[2];
           "Model_DB".w1_4[#i]:="Model_DB".w1_4[#i]+#n_m*#e[#i]*#x_m[3];
           "Model_DB".w1_5[#i]:="Model_DB".w1_5[#i]+#n_m*#e[#i]*#x_m[4];
           "Model_DB".w1_6[#i]:="Model_DB".w1_6[#i]+#n_m*#e[#i]*#x_m[5];
           "Model_DB".bias[#i]:="Model_DB".bias[#i]+#n_m*#e[#i];
       END_FOR;

       FOR #i:=0 TO "Model_DB".N-1 DO                                                
           "Model_DB".w_2[#i]:="Model_DB".w_2[#i]+#n_m*#e2*#o[#i];
       END_FOR;
           "Model_DB".bias2:="Model_DB".bias2+#n_m*#e2;
     END_FOR;

     #error_ep_m:=0.0;
     #s2:=0.0;
     FOR #long:=0 TO 249 DO

       IF #long=0 THEN
         #x_m[2]:=0.0;         // x(k-2)
         #x_m[1]:=0.0;         // x(k-1)
         #x_m[0]:="Measurement_DB".r_array[#long];  // x(k)
         #x_m[5]:=0.0;         // y(k-3)
         #x_m[4]:=0.0;         // y(k-2)
         #x_m[3]:=0.0;         // y(k-1) 
       ELSE
         #x_m[2]:=#x_m[1];     // x(k-2)
         #x_m[1]:=#x_m[0];     // x(k-1)
         #x_m[0]:="Measurement_DB".r_array[#long];  // x(k)
         #x_m[5]:=#x_m[4];     // y(k-3)             
         #x_m[4]:=#x_m[3];     // y(k-2)
         #x_m[3]:=#s2;         // y(k-1)
       END_IF;

       FOR #i:=0 TO "Model_DB".N-1 DO
          #s[#i]:=#x_m[0]*"Model_DB".w1_1[#i] + #x_m[1]*"Model_DB".w1_2[#i] + #x_m[2]*"Model_DB".w1_3[#i] + #x_m[3]*"Model_DB".w1_4[#i]; 
          #s[#i]:=#s[#i] + #x_m[4]*"Model_DB".w1_5[#i] + #x_m[5]*"Model_DB".w1_6[#i] + "Model_DB".bias[#i];
          #o[#i]:=(1.0-EXP(-#s[#i]))/(1.0+EXP(-#s[#i]));
       END_FOR;

       #s2:=0.0;
       FOR #i:=0 TO "Model_DB".N-1 DO
         #s2:=#s2+#o[#i]*"Model_DB".w_2[#i];
       END_FOR;
       #s2:=#s2+"Model_DB".bias2; 

       #e2:="Measurement_DB".y_array[#long]-#s2;                               
       #error_ep_m:=#error_ep_m+ABS(#e2);                
     END_FOR;

     IF #error_ep_m<#error_stop_m                
     THEN #stop_m:=true;                         
     ELSE #stop_m:=false;
     END_IF;

   END_IF;

   IF #training_i=true THEN           
     FOR #long := 0 TO 249 DO   
       IF #long=0 THEN          
         #x_i[2]:=0.0;             // y(k-2)
         #x_i[1]:=0.0;             // y(k-1)
         #x_i[0]:="Measurement_DB".y_array[#long]; // y(k)
         #x_i[5]:=0.0;             // x(k-3)
         #x_i[4]:=0.0;             // x(k-2)
         #x_i[3]:=0.0;             // x(k-1)
       ELSE
         #x_i[2]:=#x_i[1];         // y(k-2)
         #x_i[1]:=#x_i[0];         // y(k-1)
         #x_i[0]:="Measurement_DB".y_array[#long]; // y(k)
         #x_i[5]:=#x_i[4];         // x(k-3)
         #x_i[4]:=#x_i[3];         // x(k-2)
         #x_i[3]:="Measurement_DB".r_array[#long-1];  // x(k-1)
       END_IF;


       FOR #i:=0 TO "Inversion_DB".N-1 DO
          #s[#i]:=#x_i[0]*"Inversion_DB".w1_1[#i] + #x_i[1]*"Inversion_DB".w1_2[#i] + #x_i[2]*"Inversion_DB".w1_3[#i] + #x_i[3]*"Inversion_DB".w1_4[#i];
          #s[#i]:=#s[#i] + #x_i[4]*"Inversion_DB".w1_5[#i] + #x_i[5]*"Inversion_DB".w1_6[#i] + "Inversion_DB".bias[#i];
          #o[#i]:=(1.0-EXP(-#s[#i]))/(1.0+EXP(-#s[#i]));
       END_FOR;

       #s2:=0.0;
       FOR #i:=0 TO "Inversion_DB".N-1 DO
           #s2:=#s2+#o[#i]*"Inversion_DB".w_2[#i];
       END_FOR;
       #s2:=#s2+"Inversion_DB".bias2;   

       #e2:="Measurement_DB".r_array[#long]-#s2;                          

       FOR #i:=0 TO "Inversion_DB".N-1 DO 
           #e[#i]:=#e2*"Inversion_DB".w_2[#i]*(1.0-#o[#i]*#o[#i]);// gdzie f'(s)=1-o(i)*o(i)
       END_FOR;

       FOR #i:=0 TO "Inversion_DB".N-1 DO                                              
           "Inversion_DB".w1_1[#i]:="Inversion_DB".w1_1[#i]+#n_i*#e[#i]*#x_i[0];
           "Inversion_DB".w1_2[#i]:="Inversion_DB".w1_2[#i]+#n_i*#e[#i]*#x_i[1];
           "Inversion_DB".w1_3[#i]:="Inversion_DB".w1_3[#i]+#n_i*#e[#i]*#x_i[2];
           "Inversion_DB".w1_4[#i]:="Inversion_DB".w1_4[#i]+#n_i*#e[#i]*#x_i[3];
           "Inversion_DB".w1_5[#i]:="Inversion_DB".w1_5[#i]+#n_i*#e[#i]*#x_i[4];
           "Inversion_DB".w1_6[#i]:="Inversion_DB".w1_6[#i]+#n_i*#e[#i]*#x_i[5];
           "Inversion_DB".bias[#i]:="Inversion_DB".bias[#i]+#n_i*#e[#i];
       END_FOR;

       FOR #i:=0 TO "Inversion_DB".N-1 DO                                                 
           "Inversion_DB".w_2[#i]:="Inversion_DB".w_2[#i]+#n_i*#e2*#o[#i];
       END_FOR;
           "Inversion_DB".bias2:="Inversion_DB".bias2+#n_i*#e2;
     END_FOR;

     #error_ep_i:=0.0;
     #s2:=0.0;
     FOR #long := 0 TO 249 DO   

       IF #long=0 THEN
         #x_i[2]:=0.0;             // y(k-2)
         #x_i[1]:=0.0;             // y(k-1)
         #x_i[0]:="Measurement_DB".y_array[#long]; // y(k)
         #x_i[5]:=0.0;             // x(k-3)
         #x_i[4]:=0.0;             // x(k-2)
         #x_i[3]:=0.0;             // x(k-1)
       ELSE
         #x_i[2]:=#x_i[1];         // y(k-2)
         #x_i[1]:=#x_i[0];         // y(k-1)
         #x_i[0]:="Measurement_DB".y_array[#long]; // y(k)
         #x_i[5]:=#x_i[4];         // x(k-3)
         #x_i[4]:=#x_i[3];         // x(k-2)
         #x_i[3]:=#s2;             // x(k-1)
       END_IF;

       FOR #i:=0 TO "Inversion_DB".N-1 DO  
          #s[#i]:=#x_i[0]*"Inversion_DB".w1_1[#i] + #x_i[1]*"Inversion_DB".w1_2[#i] + #x_i[2]*"Inversion_DB".w1_3[#i] + #x_i[3]*"Inversion_DB".w1_4[#i] + #x_i[4]*"Inversion_DB".w1_5[#i] + #x_i[5]*"Inversion_DB".w1_6[#i] + "Inversion_DB".bias[#i];
          #o[#i]:=(1.0-EXP(-#s[#i]))/(1.0+EXP(-#s[#i]));
       END_FOR;

       #s2:=0.0;
       FOR #i:=0 TO "Inversion_DB".N-1 DO  
           #s2:=#s2+#o[#i]*"Inversion_DB".w_2[#i];
       END_FOR;
       #s2:=#s2+"Inversion_DB".bias2;      

       #e2:="Measurement_DB".r_array[#long]-#s2;                                   
       #error_ep_i:=#error_ep_i+ABS(#e2);             
     END_FOR;

     IF #error_ep_i<#error_stop_i                      
     THEN #stop_i:=true;                           
     ELSE #stop_i:=false;
     END_IF;

   END_IF;


   IF #epoch=(#epoch_stop_m-1)          
   THEN #stop_m:=true;
   END_IF;
   IF #epoch=(#epoch_stop_i-1)        
   THEN #stop_i:=true;
   END_IF;
   #epoch:=#epoch+1.0;
END_FUNCTION_BLOCK

FUNCTION_BLOCK "Model"   // FB3, SCL
{ S7_Optimized_Access := 'FALSE' }
VERSION : 0.1
   VAR_INPUT
      wejscie : Real;   // wejscie modelu
   END_VAR
   VAR_OUTPUT
      wyjscie : Real;   // wyjscie modelu
   END_VAR
   VAR
      x : Array[0..5] of Real;   // tablica wejść sieci
      s : Array[0..7] of Real;   // tablica sum ważonych neuronów warstwy ukrytej
      o : Array[0..7] of Real;   // tablica wyjść neuronów warstwy ukrytej
      s2 : Real;   // suma ważona warstwy wyjściowej
      i : Int;   // zmienna pomocnicza
      w1_1 : Array[0..7] of Real;   // wagi połączenia 1 wejscia z neuronami w. ukrytej
      w1_2 : Array[0..7] of Real;   // wagi połączenia 2 wejscia z neuronami w. ukrytej
      w1_3 : Array[0..7] of Real;   // wagi połączenia 3 wejscia z neuronami w. ukrytej
      w1_4 : Array[0..7] of Real;   // wagi połączenia 4 wejscia z neuronami w. ukrytej
      w1_5 : Array[0..7] of Real;   // wagi połączenia 5 wejscia z neuronami w. ukrytej
      w1_6 : Array[0..7] of Real;   // wagi połączenia 6 wejscia z neuronami w. ukrytej
      w_2 : Array[0..7] of Real;   // wagi połączenia neuronów w.ukrytej z neuronem wyjsciowym
      bias : Array[0..7] of Real;   // tablica biasów warstwy ukrytej
      bias2 : Real;   // bias warstwy wyjściowej
      N : Int;   // liczba neuronów w warstwie ukrytej
   END_VAR
BEGIN
   #x[2]:=#x[1];             // x(k-2)
   #x[1]:=#x[0];             // x(k-1)
   #x[0]:=#wejscie;          // x(k)
   #x[5]:=#x[4];             // y(k-3)
   #x[4]:=#x[3];             // y(k-2)
   #x[3]:=#s2;               // y(k-1)

   FOR #i:=0 TO #N-1 DO
      #s[#i]:=#x[0]*#w1_1[#i] + #x[1]*#w1_2[#i] + #x[2]*#w1_3[#i];
      #s[#i]:=#s[#i] + #x[3]*#w1_4[#i] + #x[4]*#w1_5[#i] + #x[5]*#w1_6[#i] + #bias[#i]; // jw, + bias
      #o[#i]:=(1.0-EXP(-#s[#i]))/(1.0+EXP(-#s[#i])); //f. activation sigmoidalna
    END_FOR;

   #s2:=0.0;
   FOR #i:=0 TO #N-1 DO 
       #s2:=#s2+#o[#i]*#w_2[#i];
   END_FOR;

   #s2:=#s2+#bias2;
   #wyjscie:=#s2;
END_FUNCTION_BLOCK

FUNCTION_BLOCK "Inversion"   // FB4, SCL
{ S7_Optimized_Access := 'FALSE' }
VERSION : 0.1
   VAR_INPUT
      wejscie : Real;
   END_VAR
   VAR_OUTPUT
      wyjscie : Real;
   END_VAR
   VAR
      x : Array[0..5] of Real;
      s : Array[0..7] of Real;
      o : Array[0..7] of Real;
      s2 : Real;
      i : Int;
      w1_1 : Array[0..7] of Real;
      w1_2 : Array[0..7] of Real;
      w1_3 : Array[0..7] of Real;
      w1_4 : Array[0..7] of Real;
      w1_5 : Array[0..7] of Real;
      w1_6 : Array[0..7] of Real;
      w_2 : Array[0..7] of Real;
      bias : Array[0..7] of Real;
      bias2 : Real;
      N : Int;
   END_VAR
BEGIN
   #x[2]:=#x[1];             // x(k-2)
   #x[1]:=#x[0];             // x(k-1)
   #x[0]:=#wejscie;          // x(k)
   #x[5]:=#x[4];             // y(k-3)
   #x[4]:=#x[3];             // y(k-2)
   #x[3]:=#s2;               // y(k-1)

   FOR #i:=0 TO #N-1 DO
      #s[#i]:=#x[0]*#w1_1[#i] + #x[1]*#w1_2[#i] + #x[2]*#w1_3[#i];
      #s[#i]:=#s[#i] + #x[3]*#w1_4[#i] + #x[4]*#w1_5[#i] + #x[5]*#w1_6[#i] + #bias[#i]; // jw, + bias
      #o[#i]:=(1.0-EXP(-#s[#i]))/(1.0+EXP(-#s[#i])); // f. sigmoidalna
    END_FOR;

   #s2:=0.0;
   FOR #i:=0 TO #N-1 DO
       #s2:=#s2+#o[#i]*#w_2[#i];
   END_FOR;

   #s2:=#s2+#bias2;
   #wyjscie:=#s2;
END_FUNCTION_BLOCK

FUNCTION_BLOCK "IMC+PID"   // FB5, SCL
{ S7_Optimized_Access := 'FALSE' }
VERSION : 0.1
   VAR_INPUT
      SP : Real;   // wartosc zadana
      PV : Real;   // odpowiedz obiektu
   END_VAR
   VAR_OUTPUT
      MV : Real;   // sygnał sterujący
   END_VAR
   VAR
      PV_model : Real;   // odpowiedz modelu
      e_ob_mo : Real;   // roznica obiekt - model
      "e" : Real;   // SP - e_ob_mo
      ef : Array[0..1] of Real;   // tablica, filtr + chwila poprzednia
      MV1 : Real;   // syg. sterujacy z inwersji
      MV2 : Real;   // syg. sterujacy z PID
   END_VAR
BEGIN
   "Model_DB"(wejscie:=#MV,
              wyjscie=>#PV_model);


   #e_ob_mo:=#PV-#PV_model;
   #e:=#SP-#e_ob_mo;

   #ef[1]:=#ef[0];
   #ef[0]:=0.2835*#e+0.7165*#ef[1];


   "Inversion_DB"(wejscie:=#ef[0],
                 wyjscie=>#MV1);

   "PID_DB_1"(SP:=#SP,
              PV:=#PV,
              MV:=#MV,
              kp:=0.2,
              ki:=0.8,
              kd:=0.1,
              MV_PID=>#MV2);


   #MV:=#MV1+#MV2;

   IF #MV>10.0 THEN
       #MV:=10.0;
   END_IF;

   IF #MV<-10.0 THEN
       #MV:=-10.0;
   END_IF;
END_FUNCTION_BLOCK

FUNCTION_BLOCK "Generator"   // FB15, SCL
{ S7_Optimized_Access := 'FALSE' }
VERSION : 0.1
   VAR_OUTPUT
      wartosc_zaklocenia : Real;
      u : LReal;
   END_VAR
   VAR
      k : Real;
      i : Int;
   END_VAR
BEGIN
   (*SV*)
   IF #k<=25.0 THEN
   #u:=0.0; 
   END_IF;
   IF #k>25.0 THEN
   #u:=2.0; 
   END_IF;
   IF #k>175.0 THEN
   #u:=-2.0; 
   END_IF;
   IF #k>250.0 THEN
   #u:=2.0*SIN(2.0*3.1416*#k/50.0); 
   END_IF;
   IF #k>400.0 THEN
   #u:=0.0; 
   END_IF;

   (*ZAKLOCENIE*)
   IF #k<=100.0 THEN
   #wartosc_zaklocenia:=0.0; 
   END_IF;
   IF #k>75.0 THEN
   #wartosc_zaklocenia:=-1.0; 
   END_IF;
   IF #k>125.0 THEN
   #wartosc_zaklocenia:=0.0; 
   END_IF;
   IF #k>300.0 THEN
   #wartosc_zaklocenia:=-1.0; 
   END_IF;
   IF #k>400.0 THEN
   #wartosc_zaklocenia:=0.0; 
   END_IF;

   #k:=#k+1.0;
END_FUNCTION_BLOCK

FUNCTION_BLOCK "Object"   // FB30, SCL
{ S7_Optimized_Access := 'FALSE' }
VERSION : 0.1
   VAR_INPUT
      r : Real;
      disruption : Real;
   END_VAR
   VAR_OUTPUT
      y : Real;
   END_VAR
   VAR
      x_array : Array[0..2] of Real;
      y_array : Array[0..2] of Real;
   END_VAR
BEGIN
   #x_array[2]:=#x_array[1];
   #x_array[1]:=#x_array[0];
   #x_array[0]:=#r;

   #y_array[2]:=#y_array[1];
   #y_array[1]:=#y_array[0];


   #y_array[0]:=0.3*1.3*#x_array[0]+0.1*#x_array[1]+0.6*0.8*#y_array[1]-0.4*1.5*#y_array[2]+0.03*0.5*#y_array[2]*#y_array[2] + #disruption;


   IF ABS(#y_array[0])<0.0001 THEN
     #y_array[0]:=0.0;
   END_IF;

   #y:=#y_array[0];
END_FUNCTION_BLOCK

FUNCTION "StartupValues" : Void   // FC1, SCL
{ S7_Optimized_Access := 'FALSE' }
VERSION : 0.1
BEGIN
   "Model_DB".N:=8;
   "Inversion_DB".N:=8;

   "Model_DB".w1_1[0]:=0.0947;"Model_DB".w1_1[1]:=-0.0755;"Model_DB".w1_1[2]:=-0.0989;"Model_DB".w1_1[3]:=-0.0972;"Model_DB".w1_1[4]:=0.0946;"Model_DB".w1_1[5]:=-0.0280;"Model_DB".w1_1[6]:=-0.0111;"Model_DB".w1_1[7]:=-0.0137;
   "Model_DB".w1_2[0]:=-0.0590;"Model_DB".w1_2[1]:=-0.0059;"Model_DB".w1_2[2]:=0.0382;"Model_DB".w1_2[3]:=-0.0107;"Model_DB".w1_2[4]:=-0.0165;"Model_DB".w1_2[5]:=-0.0539;"Model_DB".w1_2[6]:=0.0721;"Model_DB".w1_2[7]:=0.0880;
   "Model_DB".w1_3[0]:=-0.0367;"Model_DB".w1_3[1]:=0.0941;"Model_DB".w1_3[2]:=0.0776;"Model_DB".w1_3[3]:=0.0644;"Model_DB".w1_3[4]:=0.0289;"Model_DB".w1_3[5]:=0.0670;"Model_DB".w1_3[6]:=-0.0905;"Model_DB".w1_3[7]:=0.0183;
   "Model_DB".w1_4[0]:=0.0985;"Model_DB".w1_4[1]:=-0.0487;"Model_DB".w1_4[2]:=-0.0788;"Model_DB".w1_4[3]:=-0.0514;"Model_DB".w1_4[4]:=-0.0354;"Model_DB".w1_4[5]:=0.0116;"Model_DB".w1_4[6]:=-0.0407;"Model_DB".w1_4[7]:=0.0417;
   "Model_DB".w1_5[0]:=-0.0128;"Model_DB".w1_5[1]:=0.0692;"Model_DB".w1_5[2]:=-0.0502;"Model_DB".w1_5[3]:=0.0642;"Model_DB".w1_5[4]:=0.0651;"Model_DB".w1_5[5]:=-0.0490;"Model_DB".w1_5[6]:=0.0467;"Model_DB".w1_5[7]:=0.0328;
   "Model_DB".w1_6[0]:=0.0572;"Model_DB".w1_6[1]:=0.0508;"Model_DB".w1_6[2]:=0.0995;"Model_DB".w1_6[3]:=0.0541;"Model_DB".w1_6[4]:=0.0762;"Model_DB".w1_6[5]:=-0.0299;"Model_DB".w1_6[6]:=0.0620;"Model_DB".w1_6[7]:=0.0941;

   "Model_DB".w_2[0]:=-0.0526;"Model_DB".w_2[1]:=-0.0155;"Model_DB".w_2[2]:=0.0993;"Model_DB".w_2[3]:=0.0224;"Model_DB".w_2[4]:=-0.0963;"Model_DB".w_2[5]:=0.0916;"Model_DB".w_2[6]:=-0.0890;"Model_DB".w_2[7]:=0.0937;

   "Model_DB".bias[0]:=-0.0168;"Model_DB".bias[1]:=0.0702;"Model_DB".bias[2]:=0.0775;"Model_DB".bias[3]:=-0.0036;"Model_DB".bias[4]:=-0.0820;"Model_DB".bias[5]:=-0.0017;"Model_DB".bias[6]:=0.0254;"Model_DB".bias[7]:=0.0210;
   "Model_DB".bias2:=0.0159;

   "Inversion_DB".w1_1[0]:=0.0502;"Inversion_DB".w1_1[1]:=-0.0982;"Inversion_DB".w1_1[2]:=-0.0046;"Inversion_DB".w1_1[3]:=-0.0499;"Inversion_DB".w1_1[4]:=-0.0384;"Inversion_DB".w1_1[5]:=0.0934;"Inversion_DB".w1_1[6]:=-0.0582;"Inversion_DB".w1_1[7]:=0.0041;
   "Inversion_DB".w1_2[0]:=-0.0549;"Inversion_DB".w1_2[1]:=0.0134;"Inversion_DB".w1_2[2]:=0.0996;"Inversion_DB".w1_2[3]:=-0.0736;"Inversion_DB".w1_2[4]:=0.0909;"Inversion_DB".w1_2[5]:=-0.0752;"Inversion_DB".w1_2[6]:=-0.0628;"Inversion_DB".w1_2[7]:=0.0293;
   "Inversion_DB".w1_3[0]:=-0.0744;"Inversion_DB".w1_3[1]:=-0.0837;"Inversion_DB".w1_3[2]:=0.0318;"Inversion_DB".w1_3[3]:=-0.0945;"Inversion_DB".w1_3[4]:=0.0970;"Inversion_DB".w1_3[5]:=0.0079;"Inversion_DB".w1_3[6]:=-0.0252;"Inversion_DB".w1_3[7]:=0.0413;
   "Inversion_DB".w1_4[0]:=0.0895;"Inversion_DB".w1_4[1]:=-0.0235;"Inversion_DB".w1_4[2]:=0.0386;"Inversion_DB".w1_4[3]:=0.0204;"Inversion_DB".w1_4[4]:=0.0551;"Inversion_DB".w1_4[5]:=0.0184;"Inversion_DB".w1_4[6]:=-0.0248;"Inversion_DB".w1_4[7]:=0.0701;
   "Inversion_DB".w1_5[0]:=-0.0549;"Inversion_DB".w1_5[1]:=0.0594;"Inversion_DB".w1_5[2]:=0.0994;"Inversion_DB".w1_5[3]:=-0.0437;"Inversion_DB".w1_5[4]:=0.0421;"Inversion_DB".w1_5[5]:=0.0329;"Inversion_DB".w1_5[6]:=-0.0170;"Inversion_DB".w1_5[7]:=-0.0003;
   "Inversion_DB".w1_6[0]:=0.0898;"Inversion_DB".w1_6[1]:=0.0906;"Inversion_DB".w1_6[2]:=0.0466;"Inversion_DB".w1_6[3]:=-0.0231;"Inversion_DB".w1_6[4]:=-0.0920;"Inversion_DB".w1_6[5]:=0.0166;"Inversion_DB".w1_6[6]:=0.0129;"Inversion_DB".w1_6[7]:=-0.0290;

   "Inversion_DB".w_2[0]:=0.0760;"Inversion_DB".w_2[1]:=0.0249;"Inversion_DB".w_2[2]:=0.0248;"Inversion_DB".w_2[3]:=-0.0409;"Inversion_DB".w_2[4]:=-0.0851;"Inversion_DB".w_2[5]:=-0.0413;"Inversion_DB".w_2[6]:=-0.0531;"Inversion_DB".w_2[7]:=-0.0308;

   "Inversion_DB".bias[0]:=0.0697;"Inversion_DB".bias[1]:=-0.0679;"Inversion_DB".bias[2]:=-0.0684;"Inversion_DB".bias[3]:=0.0017;"Inversion_DB".bias[4]:=0.0207;"Inversion_DB".bias[5]:=-0.0677;"Inversion_DB".bias[6]:=0.0271;"Inversion_DB".bias[7]:=0.0688;
   "Inversion_DB".bias2:=0.0565;

   "Measurement_DB".r_array[0]:=7.7353;"Measurement_DB".r_array[1]:=-1.5888;"Measurement_DB".r_array[2]:=-4.3230;"Measurement_DB".r_array[3]:=-9.0364;"Measurement_DB".r_array[4]:=-5.6167;
   "Measurement_DB".r_array[5]:=-5.2165;"Measurement_DB".r_array[6]:=-9.4148;"Measurement_DB".r_array[7]:=4.0462;"Measurement_DB".r_array[8]:=-9.8473;"Measurement_DB".r_array[9]:=2.2184;
   "Measurement_DB".r_array[10]:=-1.8382;"Measurement_DB".r_array[11]:=-5.0211;"Measurement_DB".r_array[12]:=3.0492;"Measurement_DB".r_array[13]:=-3.5945;"Measurement_DB".r_array[14]:=-7.9266;
   "Measurement_DB".r_array[15]:=0.7113;"Measurement_DB".r_array[16]:=-6.7026;"Measurement_DB".r_array[17]:=7.6688;"Measurement_DB".r_array[18]:=3.3291;"Measurement_DB".r_array[19]:=6.9548;
   "Measurement_DB".r_array[20]:=5.2532;"Measurement_DB".r_array[21]:=6.1403;"Measurement_DB".r_array[22]:=2.6590;"Measurement_DB".r_array[23]:=4.2085;"Measurement_DB".r_array[24]:=3.7733;
   "Measurement_DB".r_array[25]:=-3.5810;"Measurement_DB".r_array[26]:=0.6330;"Measurement_DB".r_array[27]:=7.4639;"Measurement_DB".r_array[28]:=-8.9092;"Measurement_DB".r_array[29]:=0.0080;
   "Measurement_DB".r_array[30]:=-1.3447;"Measurement_DB".r_array[31]:=8.0856;"Measurement_DB".r_array[32]:=2.6037;"Measurement_DB".r_array[33]:=9.6607;"Measurement_DB".r_array[34]:=1.7040;
   "Measurement_DB".r_array[35]:=6.8127;"Measurement_DB".r_array[36]:=-0.6237;"Measurement_DB".r_array[37]:=0.9044;"Measurement_DB".r_array[38]:=-6.4179;"Measurement_DB".r_array[39]:=2.6892;
   "Measurement_DB".r_array[40]:=9.2592;"Measurement_DB".r_array[41]:=0.6803;"Measurement_DB".r_array[42]:=-0.4077;"Measurement_DB".r_array[43]:=5.8733;"Measurement_DB".r_array[44]:=-8.1457;
   "Measurement_DB".r_array[45]:=7.6160;"Measurement_DB".r_array[46]:=-9.9225;"Measurement_DB".r_array[47]:=0.2306;"Measurement_DB".r_array[48]:=3.5693;"Measurement_DB".r_array[49]:=1.3150;
   "Measurement_DB".r_array[50]:=-0.4308;"Measurement_DB".r_array[51]:=-3.5897;"Measurement_DB".r_array[52]:=2.0316;"Measurement_DB".r_array[53]:=8.2631;"Measurement_DB".r_array[54]:=3.6504;
   "Measurement_DB".r_array[55]:=8.9347;"Measurement_DB".r_array[56]:=-8.0182;"Measurement_DB".r_array[57]:=0.2206;"Measurement_DB".r_array[58]:=-7.7974;"Measurement_DB".r_array[59]:=0.9052;
   "Measurement_DB".r_array[60]:=3.7757;"Measurement_DB".r_array[61]:=-7.0517;"Measurement_DB".r_array[62]:=5.5512;"Measurement_DB".r_array[63]:=-2.0190;"Measurement_DB".r_array[64]:=7.9660;
   "Measurement_DB".r_array[65]:=-3.8591;"Measurement_DB".r_array[66]:=-8.7790;"Measurement_DB".r_array[67]:=-5.6106;"Measurement_DB".r_array[68]:=-8.3433;"Measurement_DB".r_array[69]:=9.0079;
   "Measurement_DB".r_array[70]:=-9.6726;"Measurement_DB".r_array[71]:=-7.7066;"Measurement_DB".r_array[72]:=-9.7518;"Measurement_DB".r_array[73]:=-5.6755;"Measurement_DB".r_array[74]:=-9.7714;
   "Measurement_DB".r_array[75]:=2.8490;"Measurement_DB".r_array[76]:=0.3398;"Measurement_DB".r_array[77]:=-5.0892;"Measurement_DB".r_array[78]:=-6.1251;"Measurement_DB".r_array[79]:=-8.1826;
   "Measurement_DB".r_array[80]:=-2.6312;"Measurement_DB".r_array[81]:=-9.8441;"Measurement_DB".r_array[82]:=2.0540;"Measurement_DB".r_array[83]:=-0.4229;"Measurement_DB".r_array[84]:=-3.8376;
   "Measurement_DB".r_array[85]:=4.8889;"Measurement_DB".r_array[86]:=6.7870;"Measurement_DB".r_array[87]:=-4.7514;"Measurement_DB".r_array[88]:=0.2848;"Measurement_DB".r_array[89]:=-1.0645;
   "Measurement_DB".r_array[90]:=-3.1758;"Measurement_DB".r_array[91]:=6.7828;"Measurement_DB".r_array[92]:=9.6499;"Measurement_DB".r_array[93]:=2.5293;"Measurement_DB".r_array[94]:=-6.3745;
   "Measurement_DB".r_array[95]:=-7.5397;"Measurement_DB".r_array[96]:=1.5994;"Measurement_DB".r_array[97]:=-3.4293;"Measurement_DB".r_array[98]:=-4.6363;"Measurement_DB".r_array[99]:=1.0048;
   "Measurement_DB".r_array[100]:=-6.3897;"Measurement_DB".r_array[101]:=3.5698;"Measurement_DB".r_array[102]:=-8.8862;"Measurement_DB".r_array[103]:=-9.3189;"Measurement_DB".r_array[104]:=-4.2696;
   "Measurement_DB".r_array[105]:=-8.4522;"Measurement_DB".r_array[106]:=8.0114;"Measurement_DB".r_array[107]:=6.9321;"Measurement_DB".r_array[108]:=-2.0860;"Measurement_DB".r_array[109]:=-6.6157;
   "Measurement_DB".r_array[110]:=-1.3910;"Measurement_DB".r_array[111]:=-1.6756;"Measurement_DB".r_array[112]:=4.5753;"Measurement_DB".r_array[113]:=-1.8705;"Measurement_DB".r_array[114]:=9.0361;
   "Measurement_DB".r_array[115]:=8.2397;"Measurement_DB".r_array[116]:=9.0283;"Measurement_DB".r_array[117]:=-3.0800;"Measurement_DB".r_array[118]:=-4.1951;"Measurement_DB".r_array[119]:=7.7340;
   "Measurement_DB".r_array[120]:=-5.7994;"Measurement_DB".r_array[121]:=-7.3825;"Measurement_DB".r_array[122]:=0.4103;"Measurement_DB".r_array[123]:=8.1093;"Measurement_DB".r_array[124]:=-1.9494;
   "Measurement_DB".r_array[125]:=-5.6848;"Measurement_DB".r_array[126]:=-8.4252;"Measurement_DB".r_array[127]:=8.6612;"Measurement_DB".r_array[128]:=2.0574;"Measurement_DB".r_array[129]:=-2.4502;
   "Measurement_DB".r_array[130]:=3.2986;"Measurement_DB".r_array[131]:=5.8438;"Measurement_DB".r_array[132]:=-3.3302;"Measurement_DB".r_array[133]:=3.8532;"Measurement_DB".r_array[134]:=-5.9237;
   "Measurement_DB".r_array[135]:=9.1743;"Measurement_DB".r_array[136]:=4.2366;"Measurement_DB".r_array[137]:=-6.6619;"Measurement_DB".r_array[138]:=-1.1445;"Measurement_DB".r_array[139]:=2.6599;
   "Measurement_DB".r_array[140]:=8.5993;"Measurement_DB".r_array[141]:=0.5866;"Measurement_DB".r_array[142]:=2.5295;"Measurement_DB".r_array[143]:=3.6164;"Measurement_DB".r_array[144]:=8.4640;
   "Measurement_DB".r_array[145]:=-6.9433;"Measurement_DB".r_array[146]:=-1.8856;"Measurement_DB".r_array[147]:=-3.7505;"Measurement_DB".r_array[148]:=3.8780;"Measurement_DB".r_array[149]:=7.8138;
   "Measurement_DB".r_array[150]:=-0.1866;"Measurement_DB".r_array[151]:=6.1165;"Measurement_DB".r_array[152]:=-3.4712;"Measurement_DB".r_array[153]:=0.9976;"Measurement_DB".r_array[154]:=-2.2243;
   "Measurement_DB".r_array[155]:=7.9366;"Measurement_DB".r_array[156]:=3.5224;"Measurement_DB".r_array[157]:=6.5679;"Measurement_DB".r_array[158]:=-7.7982;"Measurement_DB".r_array[159]:=-4.4155;
   "Measurement_DB".r_array[160]:=5.3527;"Measurement_DB".r_array[161]:=-5.6789;"Measurement_DB".r_array[162]:=-9.3188;"Measurement_DB".r_array[163]:=-1.2690;"Measurement_DB".r_array[164]:=8.7373;
   "Measurement_DB".r_array[165]:=-4.7582;"Measurement_DB".r_array[166]:=1.3949;"Measurement_DB".r_array[167]:=-2.8089;"Measurement_DB".r_array[168]:=-9.4632;"Measurement_DB".r_array[169]:=0.0084;
   "Measurement_DB".r_array[170]:=6.5403;"Measurement_DB".r_array[171]:=-4.8204;"Measurement_DB".r_array[172]:=-9.0823;"Measurement_DB".r_array[173]:=-5.0706;"Measurement_DB".r_array[174]:=3.2146;
   "Measurement_DB".r_array[175]:=-3.4118;"Measurement_DB".r_array[176]:=3.1899;"Measurement_DB".r_array[177]:=-9.7399;"Measurement_DB".r_array[178]:=4.3614;"Measurement_DB".r_array[179]:=-2.1776;
   "Measurement_DB".r_array[180]:=-9.3299;"Measurement_DB".r_array[181]:=-1.8797;"Measurement_DB".r_array[182]:=4.3262;"Measurement_DB".r_array[183]:=8.4267;"Measurement_DB".r_array[184]:=9.6803;
   "Measurement_DB".r_array[185]:=9.6684;"Measurement_DB".r_array[186]:=7.9261;"Measurement_DB".r_array[187]:=7.3141;"Measurement_DB".r_array[188]:=6.0192;"Measurement_DB".r_array[189]:=1.0996;
   "Measurement_DB".r_array[190]:=-1.6226;"Measurement_DB".r_array[191]:=-7.4575;"Measurement_DB".r_array[192]:=3.0924;"Measurement_DB".r_array[193]:=7.2793;"Measurement_DB".r_array[194]:=-4.5080;
   "Measurement_DB".r_array[195]:=6.8033;"Measurement_DB".r_array[196]:=-8.5849;"Measurement_DB".r_array[197]:=-2.4242;"Measurement_DB".r_array[198]:=-4.6366;"Measurement_DB".r_array[199]:=-6.9416;
   "Measurement_DB".r_array[200]:=2.6200;"Measurement_DB".r_array[201]:=-3.6725;"Measurement_DB".r_array[202]:=9.1822;"Measurement_DB".r_array[203]:=-0.0265;"Measurement_DB".r_array[204]:=4.7722;
   "Measurement_DB".r_array[205]:=-9.7449;"Measurement_DB".r_array[206]:=2.1071;"Measurement_DB".r_array[207]:=1.5290;"Measurement_DB".r_array[208]:=6.1476;"Measurement_DB".r_array[209]:=3.0994;
   "Measurement_DB".r_array[210]:=7.5646;"Measurement_DB".r_array[211]:=8.0475;"Measurement_DB".r_array[212]:=-6.9553;"Measurement_DB".r_array[213]:=-6.1484;"Measurement_DB".r_array[214]:=5.8195;
   "Measurement_DB".r_array[215]:=-8.7859;"Measurement_DB".r_array[216]:=-2.2035;"Measurement_DB".r_array[217]:=-4.0007;"Measurement_DB".r_array[218]:=4.6836;"Measurement_DB".r_array[219]:=-7.9158;
   "Measurement_DB".r_array[220]:=5.8515;"Measurement_DB".r_array[221]:=5.6546;"Measurement_DB".r_array[222]:=0.6480;"Measurement_DB".r_array[223]:=-4.9330;"Measurement_DB".r_array[224]:=-8.5809;
   "Measurement_DB".r_array[225]:=2.5161;"Measurement_DB".r_array[226]:=-9.5064;"Measurement_DB".r_array[227]:=-8.7592;"Measurement_DB".r_array[228]:=-7.4078;"Measurement_DB".r_array[229]:=-0.9877;
   "Measurement_DB".r_array[230]:=3.4467;"Measurement_DB".r_array[231]:=7.1222;"Measurement_DB".r_array[232]:=-0.0311;"Measurement_DB".r_array[233]:=-9.0243;"Measurement_DB".r_array[234]:=-3.7234;
   "Measurement_DB".r_array[235]:=2.8326;"Measurement_DB".r_array[236]:=5.7277;"Measurement_DB".r_array[237]:=-4.2170;"Measurement_DB".r_array[238]:=-0.0426;"Measurement_DB".r_array[239]:=6.3687;
   "Measurement_DB".r_array[240]:=1.9026;"Measurement_DB".r_array[241]:=0.7285;"Measurement_DB".r_array[242]:=-3.3825;"Measurement_DB".r_array[243]:=-1.7662;"Measurement_DB".r_array[244]:=5.8801;
   "Measurement_DB".r_array[245]:=-3.1358;"Measurement_DB".r_array[246]:=-0.7479;"Measurement_DB".r_array[247]:=-2.6435;"Measurement_DB".r_array[248]:=3.5914;"Measurement_DB".r_array[249]:=1.3556;
END_FUNCTION

FUNCTION "TrainingFunction" : Void   // FC7, LAD
TITLE = TrainingFunction
{ S7_Optimized_Access := 'TRUE' }
VERSION : 0.1
BEGIN

REGION Network 1: Call: Training
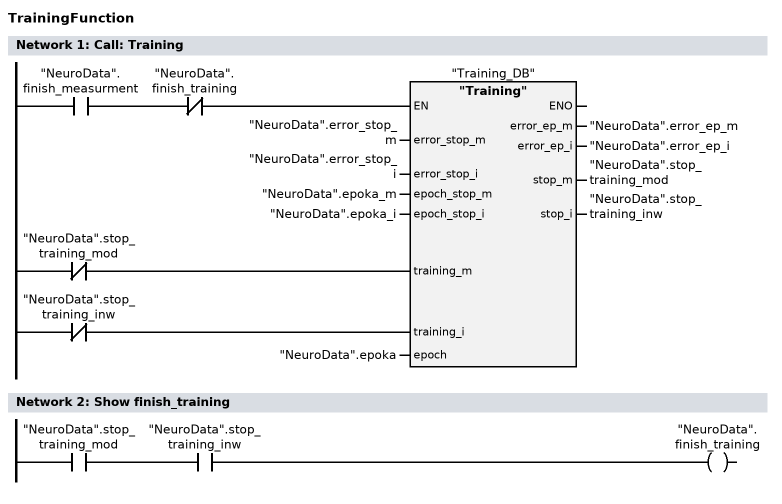
   RUNG wire#powerrail
      Contact( "NeuroData".finish_measurment )
      I_Contact( "NeuroData".finish_training )
      "Training_DB"(training_m := wire#w1, training_i := wire#w2, error_stop_m := "NeuroData".error_stop_m, error_stop_i := "NeuroData".error_stop_i, epoch_stop_m := "NeuroData".epoka_m, epoch_stop_i := "NeuroData".epoka_i, epoch := "NeuroData".epoka, error_ep_m => "NeuroData".error_ep_m, error_ep_i => "NeuroData".error_ep_i, stop_m => "NeuroData".stop_training_mod, stop_i => "NeuroData".stop_training_inw)
   END_RUNG
   RUNG wire#powerrail
      I_Contact( "NeuroData".stop_training_mod )
   END_RUNG wire#w1
   RUNG wire#powerrail
      I_Contact( "NeuroData".stop_training_inw )
   END_RUNG wire#w2
   // the same network as SCL:
   IF "NeuroData".finish_measurment AND NOT "NeuroData".finish_training THEN
       "Training_DB"(error_stop_m := "NeuroData".error_stop_m,   // "Training"
                     error_stop_i := "NeuroData".error_stop_i,
                     epoch_stop_m := "NeuroData".epoka_m,
                     epoch_stop_i := "NeuroData".epoka_i,
                     training_m := NOT "NeuroData".stop_training_mod,
                     training_i := NOT "NeuroData".stop_training_inw,
                     epoch := "NeuroData".epoka,
                     error_ep_m => "NeuroData".error_ep_m,
                     error_ep_i => "NeuroData".error_ep_i,
                     stop_m => "NeuroData".stop_training_mod,
                     stop_i => "NeuroData".stop_training_inw);
   END_IF;
END_REGION

REGION Network 2: Show finish_training
   RUNG wire#powerrail
      Contact( "NeuroData".stop_training_mod )
      Contact( "NeuroData".stop_training_inw )
      Coil( "NeuroData".finish_training )
   END_RUNG
   // the same network as SCL:
   "NeuroData".finish_training := "NeuroData".stop_training_mod AND "NeuroData".stop_training_inw;
END_REGION
END_FUNCTION

ORGANIZATION_BLOCK "NeuralNetwork"   // OB31, LAD, CyclicInterrupt
TITLE = NeuralNetwork
{ S7_Optimized_Access := 'TRUE' }
VERSION : 0.1
   VAR_INPUT
      Initial_Call : Bool;   // Initial call of this OB
      Event_Count : Int;   // Events discarded
   END_VAR
   VAR_TEMP
      MV : Real;
   END_VAR
   VAR_TEMP   // added for the SCL form of the ladder/FBD networks
      _w1 : Bool;
   END_VAR
BEGIN

REGION Network 1: Call: Measurement
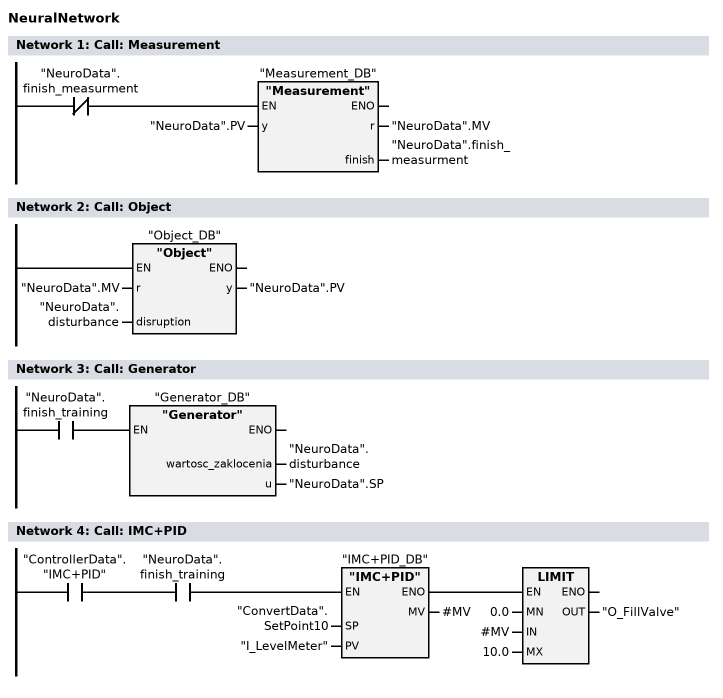
   RUNG wire#powerrail
      I_Contact( "NeuroData".finish_measurment )
      "Measurement_DB"(y := "NeuroData".PV, r => "NeuroData".MV, finish => "NeuroData".finish_measurment)
   END_RUNG
   // the same network as SCL:
   IF NOT "NeuroData".finish_measurment THEN
       "Measurement_DB"(y := "NeuroData".PV, r => "NeuroData".MV, finish => "NeuroData".finish_measurment);   // "Measurement"
   END_IF;
END_REGION

REGION Network 2: Call: Object
   RUNG wire#powerrail
      "Object_DB"(r := "NeuroData".MV, disruption := "NeuroData".disturbance, y => "NeuroData".PV)
   END_RUNG
   // the same network as SCL:
   "Object_DB"(r := "NeuroData".MV, disruption := "NeuroData".disturbance, y => "NeuroData".PV);   // "Object"
END_REGION

REGION Network 3: Call: Generator
   RUNG wire#powerrail
      Contact( "NeuroData".finish_training )
      "Generator_DB"(wartosc_zaklocenia => "NeuroData".disturbance, u => "NeuroData".SP)
   END_RUNG
   // the same network as SCL:
   IF "NeuroData".finish_training THEN
       "Generator_DB"(wartosc_zaklocenia => "NeuroData".disturbance, u => "NeuroData".SP);   // "Generator"
   END_IF;
END_REGION

REGION Network 4: Call: IMC+PID
   "IMC+PID_DB"(EN := "ControllerData"."IMC+PID" AND "NeuroData".finish_training,   // "IMC+PID"
                SP := "ConvertData".SetPoint10,
                PV := "I_LevelMeter",
                MV => #MV,
                ENO => #_w1);
   IF #_w1 THEN "O_FillValve" := LIMIT(MN := 0.0, IN := #MV, MX := 10.0); END_IF;
END_REGION
END_ORGANIZATION_BLOCK

// folder: 03_Disturbance

FUNCTION_BLOCK "RandomDisturbance"   // FB10, LAD
TITLE = RandomDisturbance
{ S7_Optimized_Access := 'TRUE' }
VERSION : 0.1
   VAR_INPUT
      DistribanceMode : Int;
      Outflow : Int;
   END_VAR
   VAR_OUTPUT
      DischargeValve : Int;
   END_VAR
   VAR
      TON_1 : TON_TIME;
      TON_2 : TON_TIME;
      TP : TP_TIME;
      TON_3 : TON_TIME;
      random : Int;
      p_Q : Bool;
   END_VAR
   VAR_TEMP   // added for the SCL form of the ladder/FBD networks
      _w1 : Bool;
   END_VAR
BEGIN

REGION Network 1: Disturbance
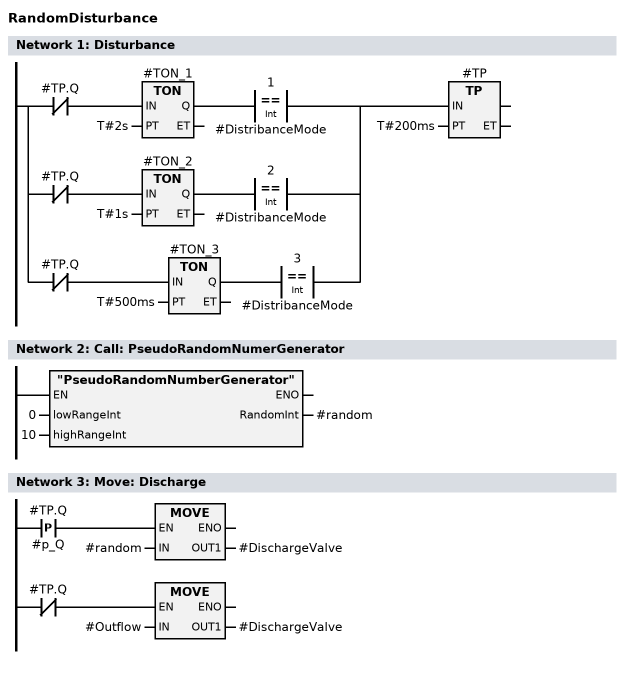
   #TON_1(IN := NOT #TP.Q, PT := T#2s);   // TON
   #TON_2(IN := NOT #TP.Q, PT := T#1s);   // TON
   #TON_3(IN := NOT #TP.Q, PT := T#500ms);   // TON
   #TP(IN := (#TON_1.Q AND (1 = #DistribanceMode)) OR (#TON_2.Q AND (2 = #DistribanceMode)) OR (#TON_3.Q AND (3 = #DistribanceMode)),   // TP
       PT := T#200ms);
END_REGION

REGION Network 2: Call: PseudoRandomNumerGenerator
   RUNG wire#powerrail
      "PseudoRandomNumberGenerator"(lowRangeInt := 0, highRangeInt := 10, RandomInt => #random)
   END_RUNG
   // the same network as SCL:
   "PseudoRandomNumberGenerator"(lowRangeInt := 0, highRangeInt := 10, RandomInt => #random);
END_REGION

REGION Network 3: Move: Discharge
   RUNG wire#powerrail
      P_Contact(operand := #TP.Q, bit := #p_Q)
      Move(in := #random, out1 => #DischargeValve)
   END_RUNG
   RUNG wire#powerrail
      I_Contact( #TP.Q )
      Move(in := #Outflow, out1 => #DischargeValve)
   END_RUNG
   // the same network as SCL:
   #_w1 := #TP.Q AND NOT #p_Q;   // rising edge of #TP.Q
   #p_Q := #TP.Q;
   IF #_w1 THEN #DischargeValve := #random; END_IF;
   IF NOT #TP.Q THEN #DischargeValve := #Outflow; END_IF;
END_REGION
END_FUNCTION_BLOCK

FUNCTION "PseudoRandomNumberGenerator" : Void   // FC4, SCL
{ S7_Optimized_Access := 'TRUE' }
VERSION : 0.1
   VAR_INPUT
      lowRangeInt : Int;
      highRangeInt : Int;
   END_VAR
   VAR_OUTPUT
      RandomInt : Int;
   END_VAR
   VAR_TEMP
      diTime : DInt;
      rTime : Real;
      timeTck : Time;
      rTemp : Real;
   END_VAR
BEGIN
    // read systemtime
   #timeTck := TIME_TCK(); // TIME

   // calculate random number
   #diTime := TIME_TO_DINT(#timeTck);
   #rTime := DINT_TO_REAL(#diTime);
   #rTemp := SIN(#rTime);

   IF #rTemp < 0 THEN
       #rTemp := #rTemp * (-1);
   END_IF;

   #RandomInt := REAL_TO_INT(#rTemp*(#highRangeInt-#lowRangeInt))+#lowRangeInt;
END_FUNCTION

FUNCTION "DisturbanceClass" : Void   // FC5, LAD
TITLE = DisturbanceClass
{ S7_Optimized_Access := 'TRUE' }
VERSION : 0.1
   VAR_TEMP
      MV : Real;
   END_VAR
BEGIN

REGION Network 1: Call: RandomDisturbance
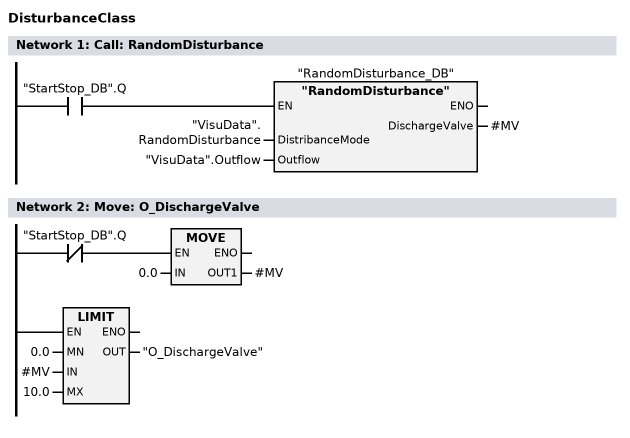
   RUNG wire#powerrail
      Contact( "StartStop_DB".Q )
      "RandomDisturbance_DB"(DistribanceMode := "VisuData".RandomDisturbance, Outflow := "VisuData".Outflow, DischargeValve => #MV)
   END_RUNG
   // the same network as SCL:
   IF "StartStop_DB".Q THEN
       "RandomDisturbance_DB"(DistribanceMode := "VisuData".RandomDisturbance,   // "RandomDisturbance"
                              Outflow := "VisuData".Outflow,
                              DischargeValve => #MV);
   END_IF;
END_REGION

REGION Network 2: Move: O_DischargeValve
   IF NOT "StartStop_DB".Q THEN #MV := 0.0; END_IF;
   "O_DischargeValve" := LIMIT(MN := 0.0, IN := #MV, MX := 10.0);
END_REGION
END_FUNCTION

(* ===== HMI "HMI_RT_1" =====
system functions are stored by id; their names below are inferred from use
connection "HMI_Connection_1": ETHERNET, SMART_S7_1500_OMS

HMI tags "00_Home"
   "Controller" : Int = PLC VisuData.Controller AT %DB1.DBW0, 1 s
   "Empty" : Bool = PLC VisuData.Empty AT %DB1.DBX0.0, 1 s
   "LowPump" : Int = PLC VisuData.LowPump AT %DB1.DBW0, 1 s
   "Outflow" : Real = PLC VisuData.Outflow AT %DB1.DBD0, 1 s
   "RandomDisturbance" : Int = PLC VisuData.RandomDisturbance AT %DB1.DBW0, 1 s
   "SetPoint" : Real = PLC VisuData.SetPoint AT %DB1.DBD0, 1 s
   "TopPump" : Int = PLC VisuData.TopPump AT %DB1.DBW0, 1 s
   "FillValve" : Real = PLC O_FillValve AT %QD30, 1 s
   "DischargeValve" : Real = PLC O_DischargeValve AT %QD34, 1 s

HMI tags "01_Settings"
   "finish_training" : Int = PLC VisuData.finish_training AT %DB1.DBW0, 1 s
   "error_stop_m" : Real = PLC NeuroData.error_stop_m AT %DB1.DBW0, 500 ms
   "error_stop_i" : Real = PLC NeuroData.error_stop_i AT %DB1.DBW0, 500 ms
   "epoch_stop_m" : Real = PLC NeuroData.epoka_m AT %DB1.DBW0, 500 ms
   "epoch_stop_i" : Real = PLC NeuroData.epoka_i AT %DB1.DBW0, 500 ms
   "epoch" : Real = PLC NeuroData.epoka AT %DB1.DBW0, 500 ms
   "rate" : Real = PLC ControllerData.rate AT %DB1.DBW0, 1 s
   "hysteresis" : Real = PLC ControllerData.hysteresis AT %DB1.DBW0, 1 s
   "kp" : Real = PLC ControllerData.kp AT %DB1.DBW0, 1 s
   "ki" : Real = PLC ControllerData.ki AT %DB1.DBW0, 1 s
   "kd" : Real = PLC ControllerData.kd AT %DB1.DBW0, 1 s
   "default" : Bool = PLC VisuData.default AT %DB1.DBX0.0, 1 s

HMI tags "00_Template"
   "Status_factoryio" : Bool = PLC VisuData.factoryio_connect AT %DB1.DBW0, 500 ms
   "Start" : Bool = PLC VisuData.Start AT %DB1.DBX0.0, 1 s
   "Stop" : Bool = PLC VisuData.Stop AT %DB1.DBX0.0, 1 s
   "SetPointShow" : Real = PLC VisuData.SetPointShow AT %DB1.DBD0, 100 ms
   "FillValveShow" : Real = PLC VisuData.FillValveShow AT %DB1.DBD0, 100 ms
   "LevelMeterShow" : Real = PLC VisuData.LevelMeterShow AT %DB1.DBD0, 100 ms
   "Status" : Bool = PLC VisuData.Status AT %DB1.DBX0.0, 500 ms

text list "Controller Type": 1 'On-Off'; 0 'Controller'; 2 'PID'; 3 'PID_Compact'; 4 'Takagi-Sugeno'; 5 'NeuralNetwork'

text list "Random Disturbance": 1 'light'; 2 'medium'; 3 'heavy'; 0 'Random Disturbance'

text list "Finish Training": 0 'No'; 1 'Yes'

screen "00_Home" 800x480, template "MyTemplate"
   GraphicView "Graphic view_2" at 136,420 size 51x41; Picture "Graphic_5"
   GraphicView "Graphic view_1" at 182,406 size 48x48; Picture "Graphic_3"
   GraphicView "Graphic view_3" at 84,420 size 54x41; Picture "Graphic_6"
   GraphicView "Graphic view_4" at 81,112 size 52x42; Picture "Graphic_7"
   GraphicView "Graphic view_5" at 25,150 size 170x275; Picture "Graphic_9"
   GraphicView "Graphic view_6" at 130,112 size 55x42; Picture "Graphic_5"
   GraphicView "Graphic view_7" at 183,97 size 48x48; Picture "Graphic_3"
   Bar "Bar_1" at 36,212 size 146x145; MinimumValue 0; MaximumValue 300
      ProcessValue <- "LevelMeterShow"
   TextField "Text field_4" at 11,44 size 55x20; Text 'Outflow'
   TextField "Text field_5" at 10,14 size 64x20; Text 'Set point'
   IOField "I/O field_2" at 80,42 size 86x27; FormatPattern 99.9; Unit  %
      ProcessValue <- "Outflow"
   Button "Button_3" at 117,327 size 53x27; TextOff 'Empty'
      on Press: SetBit("Empty")
      on Release: ResetBit("Empty")
   GraphicView "Graphic view_8" at 183,97 size 48x49; Picture "Graphic_1"
      Visibility <- "TopPump"
   GraphicView "Graphic view_9" at 182,406 size 48x49; Picture "Graphic_1"
      Visibility <- "LowPump"
   IOField "I/O field_1" at 80,12 size 86x27; FormatPattern 999.99; Unit  l
      ProcessValue <- "SetPoint"
   Button "Button_4" at 718,12 size 64x32; TextOff 'Settings'
      on Press: ActivateScreen("01_Settings", 0)
   IOField "I/O field_3" at 181,147 size 49x18; FormatPattern 99.9; Unit  %
      ProcessValue <- "FillValve"
   IOField "I/O field_4" at 182,456 size 49x18; FormatPattern 99.9; Unit  %
      ProcessValue <- "DischargeValve"
   TextField "Text field_1" at 177,14 size 94x20; Text '(0.0 - 300.0 l)'
   TextField "Text field_2" at 177,44 size 97x20; Text '(0.0 - 10.0 %)'

Template "MyTemplate" 800x480
   TextField "Text field_1" at 301,448 size 82x20; Text 'Level meter'
   TextField "Text field_2" at 447,448 size 64x20; Text 'Set point'
   TrendView "Trend view_1" at 301,55 size 484x383
   IOField "I/O field_3" at 516,443 size 42x32; FormatPattern 999; Unit  l
      ProcessValue <- "SetPointShow"
   IOField "I/O field_4" at 386,443 size 42x32; FormatPattern 999; Unit  l
      ProcessValue <- "LevelMeterShow"
   SymbolicIOField "Symbolic I/O field_1" at 301,12 size 125x32; TextOn '1'; TextOff '0'; TextList "Controller Type"
      ProcessValue <- "Controller"
   SymbolicIOField "Symbolic I/O field_2" at 440,11 size 138x33; TextOn '1'; TextOff '0'; TextList "Random Disturbance"
      ProcessValue <- "RandomDisturbance"
   TextField "Text field_3" at 576,448 size 60x20; Text 'Fill Valve'
   IOField "I/O field_5" at 637,442 size 53x32; FormatPattern 999; Unit  %
      ProcessValue <- "FillValveShow"
   Button "Button_1" at 595,12 size 53x32; TextOff 'Start'
      on Release: ResetBit("Start")
      on Press: SetBit("Start")
      Appearance <- "Status"
   Button "Button_2" at 656,12 size 53x32; TextOff 'Stop'
      on Release: ResetBit("Stop")
      on Press: SetBit("Stop")
      Appearance <- "Status"
   Rectangle "Rectangle_1" at 749,441 size 35x35
      Appearance <- "Status_factoryio"
   GraphicView "Graphic view_11" at 753,445 size 28x28; Picture "factoryIO"

screen "01_Settings" 800x480, template "MyTemplate"
   TextField "Text field_1" at 13,16 size 41x20; Text 'Ramp'
   TextField "Text field_2" at 13,57 size 36x20; Text 'Rate'
   IOField "I/O field_1" at 54,55 size 78x27; FormatPattern 99.9; Unit  r/s
      ProcessValue <- "rate"
   TextField "Text field_3" at 13,98 size 51x20; Text 'ON/OFF'
   TextField "Text field_4" at 13,139 size 43x20; Text 'Hyste'
   IOField "I/O field_2" at 63,137 size 69x27; FormatPattern 999.9
      ProcessValue <- "hysteresis"
   Button "Button_4" at 718,12 size 64x32; TextOff 'Home'
      on Press: ActivateScreen("00_Home", 0)
   TextField "Text field_9" at 159,17 size 27x20; Text 'PID'
   TextField "Text field_10" at 152,58 size 21x20; Text 'Kp'
   IOField "I/O field_5" at 202,56 size 69x27; FormatPattern 999.9
      ProcessValue <- "kp"
   TextField "Text field_11" at 152,93 size 16x20; Text 'Ki'
   IOField "I/O field_6" at 202,91 size 69x27; FormatPattern 999.9
      ProcessValue <- "ki"
   TextField "Text field_12" at 152,128 size 21x20; Text 'Kd'
   IOField "I/O field_7" at 202,126 size 69x27; FormatPattern 999.9
      ProcessValue <- "kd"
   TextField "Text field_5" at 12,179 size 104x20; Text 'Neural network'
   TextField "Text field_6" at 12,213 size 122x20; Text 'error_stop_model'
   IOField "I/O field_3" at 165,213 size 107x27; FormatPattern 999.9
      ProcessValue <- "error_stop_m"
   TextField "Text field_7" at 12,248 size 143x20; Text 'error_stop_inversion'
   TextField "Text field_14" at 11,347 size 93x20; Text 'finish training'
   TextField "Text field_15" at 12,378 size 44x20; Text 'epoch'
   IOField "I/O field_4" at 165,247 size 107x27; FormatPattern 999.9
      ProcessValue <- "error_stop_i"
   TextField "Text field_8" at 12,281 size 127x20; Text 'epoch_stop_model'
   IOField "I/O field_8" at 165,281 size 107x27; FormatPattern 999999
      ProcessValue <- "epoch_stop_m"
   TextField "Text field_13" at 12,316 size 148x20; Text 'epoch_stop_inversion'
   IOField "I/O field_9" at 164,315 size 108x27; FormatPattern 999999
      ProcessValue <- "epoch_stop_i"
   IOField "I/O field_13" at 131,381 size 141x27; FormatPattern 999999
      ProcessValue <- "epoch"
   Button "Button_1" at 13,428 size 267x32; TextOff 'Default'
      on Release: SetTag("rate", 5); SetTag("hysteresis", 2); SetTag("kp", 1); SetTag("ki", 0.1); SetTag("kd", 0.2); SetTag("epoch_stop_m", 1000); SetTag("epoch_stop_i", 2000); SetTag("error_stop_i", 5); SetTag("error_stop_m", 5)
   SymbolicIOField "Symbolic I/O field_1" at 165,347 size 110x27; TextOff '0'; TextOn '1'; TextList "Finish Training"
      ProcessValue <- "finish_training"
*)